Fanuc TP program (LS listing): S003.LS

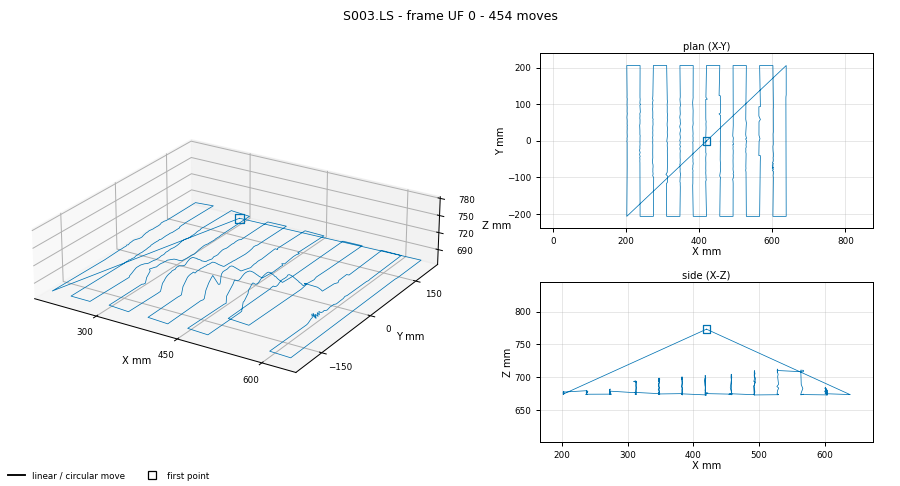
[picture p0: tool path of S003.LS in frame UF 0, 454 of 454 moves have a stored position in this frame; points joined in program order, loops and branches not executed]
/PROG  S003.LS
/ATTR
OWNER       = MNEDITOR;
COMMENT     = "";
PROG_SIZE   = 636;
CREATE      = DATE 23-01-07  TIME 11:59:14;
MODIFIED    = DATE 23-01-07  TIME 12:02:18;
FILE_NAME   = ;
VERSION     = 0;
LINE_COUNT  = 4;
MEMORY_SIZE = 992;
PROTECT     = READ_WRITE;
TCD:  STACK_SIZE    = 0,
      TASK_PRIORITY = 50,
      TIME_SLICE    = 0,
      BUSY_LAMP_OFF = 0,
      ABORT_REQUEST = 0,
      PAUSE_REQUEST = 0;
DEFAULT_GROUP    = 1,*,*,*,*;
CONTROL_CODE     = 00000000 00000000;
/MN
   1:J P[1] 100% FINE    ;
   2:L P[2] 300mm/sec CNT100    ;
   3:L P[3] 300mm/sec CNT100    ;
   4:L P[4] 300mm/sec CNT100    ;
   5:L P[5] 300mm/sec CNT100    ;
   6:L P[6] 300mm/sec CNT100    ;
   7:L P[7] 300mm/sec CNT100    ;
   8:L P[8] 300mm/sec CNT100    ;
   9:L P[9] 300mm/sec CNT100    ;
   10:L P[10] 300mm/sec CNT100    ;
   11:L P[11] 300mm/sec CNT100    ;
   12:L P[12] 300mm/sec CNT100    ;
   13:L P[13] 300mm/sec CNT100    ;
   14:L P[14] 300mm/sec CNT100    ;
   15:L P[15] 300mm/sec CNT100    ;
   16:L P[16] 300mm/sec CNT100    ;
   17:L P[17] 300mm/sec CNT100    ;
   18:L P[18] 300mm/sec CNT100    ;
   19:L P[19] 300mm/sec CNT100    ;
   20:L P[20] 300mm/sec CNT100    ;
   21:L P[21] 300mm/sec CNT100    ;
   22:L P[22] 300mm/sec CNT100    ;
   23:L P[23] 300mm/sec CNT100    ;
   24:L P[24] 300mm/sec CNT100    ;
   25:L P[25] 300mm/sec CNT100    ;
   26:L P[26] 300mm/sec CNT100    ;
   27:L P[27] 300mm/sec CNT100    ;
   28:L P[28] 300mm/sec CNT100    ;
   29:L P[29] 300mm/sec CNT100    ;
   30:L P[30] 300mm/sec CNT100    ;
   31:L P[31] 300mm/sec CNT100    ;
   32:L P[32] 300mm/sec CNT100    ;
   33:L P[33] 300mm/sec CNT100    ;
   34:L P[34] 300mm/sec CNT100    ;
   35:L P[35] 300mm/sec CNT100    ;
   36:L P[36] 300mm/sec CNT100    ;
   37:L P[37] 300mm/sec CNT100    ;
   38:L P[38] 300mm/sec CNT100    ;
   39:L P[39] 300mm/sec CNT100    ;
   40:L P[40] 300mm/sec CNT100    ;
   41:L P[41] 300mm/sec CNT100    ;
   42:L P[42] 300mm/sec CNT100    ;
   43:L P[43] 300mm/sec CNT100    ;
   44:L P[44] 300mm/sec CNT100    ;
   45:L P[45] 300mm/sec CNT100    ;
   46:L P[46] 300mm/sec CNT100    ;
   47:L P[47] 300mm/sec CNT100    ;
   48:L P[48] 300mm/sec CNT100    ;
   49:L P[49] 300mm/sec CNT100    ;
   50:L P[50] 300mm/sec CNT100    ;
   51:L P[51] 300mm/sec CNT100    ;
   52:L P[52] 300mm/sec CNT100    ;
   53:L P[53] 300mm/sec CNT100    ;
   54:L P[54] 300mm/sec CNT100    ;
   55:L P[55] 300mm/sec CNT100    ;
   56:L P[56] 300mm/sec CNT100    ;
   57:L P[57] 300mm/sec CNT100    ;
   58:L P[58] 300mm/sec CNT100    ;
   59:L P[59] 300mm/sec CNT100    ;
   60:L P[60] 300mm/sec CNT100    ;
   61:L P[61] 300mm/sec CNT100    ;
   62:L P[62] 300mm/sec CNT100    ;
   63:L P[63] 300mm/sec CNT100    ;
   64:L P[64] 300mm/sec CNT100    ;
   65:L P[65] 300mm/sec CNT100    ;
   66:L P[66] 300mm/sec CNT100    ;
   67:L P[67] 300mm/sec CNT100    ;
   68:L P[68] 300mm/sec CNT100    ;
   69:L P[69] 300mm/sec CNT100    ;
   70:L P[70] 300mm/sec CNT100    ;
   71:L P[71] 300mm/sec CNT100    ;
   72:L P[72] 300mm/sec CNT100    ;
   73:L P[73] 300mm/sec CNT100    ;
   74:L P[74] 300mm/sec CNT100    ;
   75:L P[75] 300mm/sec CNT100    ;
   76:L P[76] 300mm/sec CNT100    ;
   77:L P[77] 300mm/sec CNT100    ;
   78:L P[78] 300mm/sec CNT100    ;
   79:L P[79] 300mm/sec CNT100    ;
   80:L P[80] 300mm/sec CNT100    ;
   81:L P[81] 300mm/sec CNT100    ;
   82:L P[82] 300mm/sec CNT100    ;
   83:L P[83] 300mm/sec CNT100    ;
   84:L P[84] 300mm/sec CNT100    ;
   85:L P[85] 300mm/sec CNT100    ;
   86:L P[86] 300mm/sec CNT100    ;
   87:L P[87] 300mm/sec CNT100    ;
   88:L P[88] 300mm/sec CNT100    ;
   89:L P[89] 300mm/sec CNT100    ;
   90:L P[90] 300mm/sec CNT100    ;
   91:L P[91] 300mm/sec CNT100    ;
   92:L P[92] 300mm/sec CNT100    ;
   93:L P[93] 300mm/sec CNT100    ;
   94:L P[94] 300mm/sec CNT100    ;
   95:L P[95] 300mm/sec CNT100    ;
   96:L P[96] 300mm/sec CNT100    ;
   97:L P[97] 300mm/sec CNT100    ;
   98:L P[98] 300mm/sec CNT100    ;
   99:L P[99] 300mm/sec CNT100    ;
   100:L P[100] 300mm/sec CNT100    ;
   101:L P[101] 300mm/sec CNT100    ;
   102:L P[102] 300mm/sec CNT100    ;
   103:L P[103] 300mm/sec CNT100    ;
   104:L P[104] 300mm/sec CNT100    ;
   105:L P[105] 300mm/sec CNT100    ;
   106:L P[106] 300mm/sec CNT100    ;
   107:L P[107] 300mm/sec CNT100    ;
   108:L P[108] 300mm/sec CNT100    ;
   109:L P[109] 300mm/sec CNT100    ;
   110:L P[110] 300mm/sec CNT100    ;
   111:L P[111] 300mm/sec CNT100    ;
   112:L P[112] 300mm/sec CNT100    ;
   113:L P[113] 300mm/sec CNT100    ;
   114:L P[114] 300mm/sec CNT100    ;
   115:L P[115] 300mm/sec CNT100    ;
   116:L P[116] 300mm/sec CNT100    ;
   117:L P[117] 300mm/sec CNT100    ;
   118:L P[118] 300mm/sec CNT100    ;
   119:L P[119] 300mm/sec CNT100    ;
   120:L P[120] 300mm/sec CNT100    ;
   121:L P[121] 300mm/sec CNT100    ;
   122:L P[122] 300mm/sec CNT100    ;
   123:L P[123] 300mm/sec CNT100    ;
   124:L P[124] 300mm/sec CNT100    ;
   125:L P[125] 300mm/sec CNT100    ;
   126:L P[126] 300mm/sec CNT100    ;
   127:L P[127] 300mm/sec CNT100    ;
   128:L P[128] 300mm/sec CNT100    ;
   129:L P[129] 300mm/sec CNT100    ;
   130:L P[130] 300mm/sec CNT100    ;
   131:L P[131] 300mm/sec CNT100    ;
   132:L P[132] 300mm/sec CNT100    ;
   133:L P[133] 300mm/sec CNT100    ;
   134:L P[134] 300mm/sec CNT100    ;
   135:L P[135] 300mm/sec CNT100    ;
   136:L P[136] 300mm/sec CNT100    ;
   137:L P[137] 300mm/sec CNT100    ;
   138:L P[138] 300mm/sec CNT100    ;
   139:L P[139] 300mm/sec CNT100    ;
   140:L P[140] 300mm/sec CNT100    ;
   141:L P[141] 300mm/sec CNT100    ;
   142:L P[142] 300mm/sec CNT100    ;
   143:L P[143] 300mm/sec CNT100    ;
   144:L P[144] 300mm/sec CNT100    ;
   145:L P[145] 300mm/sec CNT100    ;
   146:L P[146] 300mm/sec CNT100    ;
   147:L P[147] 300mm/sec CNT100    ;
   148:L P[148] 300mm/sec CNT100    ;
   149:L P[149] 300mm/sec CNT100    ;
   150:L P[150] 300mm/sec CNT100    ;
   151:L P[151] 300mm/sec CNT100    ;
   152:L P[152] 300mm/sec CNT100    ;
   153:L P[153] 300mm/sec CNT100    ;
   154:L P[154] 300mm/sec CNT100    ;
   155:L P[155] 300mm/sec CNT100    ;
   156:L P[156] 300mm/sec CNT100    ;
   157:L P[157] 300mm/sec CNT100    ;
   158:L P[158] 300mm/sec CNT100    ;
   159:L P[159] 300mm/sec CNT100    ;
   160:L P[160] 300mm/sec CNT100    ;
   161:L P[161] 300mm/sec CNT100    ;
   162:L P[162] 300mm/sec CNT100    ;
   163:L P[163] 300mm/sec CNT100    ;
   164:L P[164] 300mm/sec CNT100    ;
   165:L P[165] 300mm/sec CNT100    ;
   166:L P[166] 300mm/sec CNT100    ;
   167:L P[167] 300mm/sec CNT100    ;
   168:L P[168] 300mm/sec CNT100    ;
   169:L P[169] 300mm/sec CNT100    ;
   170:L P[170] 300mm/sec CNT100    ;
   171:L P[171] 300mm/sec CNT100    ;
   172:L P[172] 300mm/sec CNT100    ;
   173:L P[173] 300mm/sec CNT100    ;
   174:L P[174] 300mm/sec CNT100    ;
   175:L P[175] 300mm/sec CNT100    ;
   176:L P[176] 300mm/sec CNT100    ;
   177:L P[177] 300mm/sec CNT100    ;
   178:L P[178] 300mm/sec CNT100    ;
   179:L P[179] 300mm/sec CNT100    ;
   180:L P[180] 300mm/sec CNT100    ;
   181:L P[181] 300mm/sec CNT100    ;
   182:L P[182] 300mm/sec CNT100    ;
   183:L P[183] 300mm/sec CNT100    ;
   184:L P[184] 300mm/sec CNT100    ;
   185:L P[185] 300mm/sec CNT100    ;
   186:L P[186] 300mm/sec CNT100    ;
   187:L P[187] 300mm/sec CNT100    ;
   188:L P[188] 300mm/sec CNT100    ;
   189:L P[189] 300mm/sec CNT100    ;
   190:L P[190] 300mm/sec CNT100    ;
   191:L P[191] 300mm/sec CNT100    ;
   192:L P[192] 300mm/sec CNT100    ;
   193:L P[193] 300mm/sec CNT100    ;
   194:L P[194] 300mm/sec CNT100    ;
   195:L P[195] 300mm/sec CNT100    ;
   196:L P[196] 300mm/sec CNT100    ;
   197:L P[197] 300mm/sec CNT100    ;
   198:L P[198] 300mm/sec CNT100    ;
   199:L P[199] 300mm/sec CNT100    ;
   200:L P[200] 300mm/sec CNT100    ;
   201:L P[201] 300mm/sec CNT100    ;
   202:L P[202] 300mm/sec CNT100    ;
   203:L P[203] 300mm/sec CNT100    ;
   204:L P[204] 300mm/sec CNT100    ;
   205:L P[205] 300mm/sec CNT100    ;
   206:L P[206] 300mm/sec CNT100    ;
   207:L P[207] 300mm/sec CNT100    ;
   208:L P[208] 300mm/sec CNT100    ;
   209:L P[209] 300mm/sec CNT100    ;
   210:L P[210] 300mm/sec CNT100    ;
   211:L P[211] 300mm/sec CNT100    ;
   212:L P[212] 300mm/sec CNT100    ;
   213:L P[213] 300mm/sec CNT100    ;
   214:L P[214] 300mm/sec CNT100    ;
   215:L P[215] 300mm/sec CNT100    ;
   216:L P[216] 300mm/sec CNT100    ;
   217:L P[217] 300mm/sec CNT100    ;
   218:L P[218] 300mm/sec CNT100    ;
   219:L P[219] 300mm/sec CNT100    ;
   220:L P[220] 300mm/sec CNT100    ;
   221:L P[221] 300mm/sec CNT100    ;
   222:L P[222] 300mm/sec CNT100    ;
   223:L P[223] 300mm/sec CNT100    ;
   224:L P[224] 300mm/sec CNT100    ;
   225:L P[225] 300mm/sec CNT100    ;
   226:L P[226] 300mm/sec CNT100    ;
   227:L P[227] 300mm/sec CNT100    ;
   228:L P[228] 300mm/sec CNT100    ;
   229:L P[229] 300mm/sec CNT100    ;
   230:L P[230] 300mm/sec CNT100    ;
   231:L P[231] 300mm/sec CNT100    ;
   232:L P[232] 300mm/sec CNT100    ;
   233:L P[233] 300mm/sec CNT100    ;
   234:L P[234] 300mm/sec CNT100    ;
   235:L P[235] 300mm/sec CNT100    ;
   236:L P[236] 300mm/sec CNT100    ;
   237:L P[237] 300mm/sec CNT100    ;
   238:L P[238] 300mm/sec CNT100    ;
   239:L P[239] 300mm/sec CNT100    ;
   240:L P[240] 300mm/sec CNT100    ;
   241:L P[241] 300mm/sec CNT100    ;
   242:L P[242] 300mm/sec CNT100    ;
   243:L P[243] 300mm/sec CNT100    ;
   244:L P[244] 300mm/sec CNT100    ;
   245:L P[245] 300mm/sec CNT100    ;
   246:L P[246] 300mm/sec CNT100    ;
   247:L P[247] 300mm/sec CNT100    ;
   248:L P[248] 300mm/sec CNT100    ;
   249:L P[249] 300mm/sec CNT100    ;
   250:L P[250] 300mm/sec CNT100    ;
   251:L P[251] 300mm/sec CNT100    ;
   252:L P[252] 300mm/sec CNT100    ;
   253:L P[253] 300mm/sec CNT100    ;
   254:L P[254] 300mm/sec CNT100    ;
   255:L P[255] 300mm/sec CNT100    ;
   256:L P[256] 300mm/sec CNT100    ;
   257:L P[257] 300mm/sec CNT100    ;
   258:L P[258] 300mm/sec CNT100    ;
   259:L P[259] 300mm/sec CNT100    ;
   260:L P[260] 300mm/sec CNT100    ;
   261:L P[261] 300mm/sec CNT100    ;
   262:L P[262] 300mm/sec CNT100    ;
   263:L P[263] 300mm/sec CNT100    ;
   264:L P[264] 300mm/sec CNT100    ;
   265:L P[265] 300mm/sec CNT100    ;
   266:L P[266] 300mm/sec CNT100    ;
   267:L P[267] 300mm/sec CNT100    ;
   268:L P[268] 300mm/sec CNT100    ;
   269:L P[269] 300mm/sec CNT100    ;
   270:L P[270] 300mm/sec CNT100    ;
   271:L P[271] 300mm/sec CNT100    ;
   272:L P[272] 300mm/sec CNT100    ;
   273:L P[273] 300mm/sec CNT100    ;
   274:L P[274] 300mm/sec CNT100    ;
   275:L P[275] 300mm/sec CNT100    ;
   276:L P[276] 300mm/sec CNT100    ;
   277:L P[277] 300mm/sec CNT100    ;
   278:L P[278] 300mm/sec CNT100    ;
   279:L P[279] 300mm/sec CNT100    ;
   280:L P[280] 300mm/sec CNT100    ;
   281:L P[281] 300mm/sec CNT100    ;
   282:L P[282] 300mm/sec CNT100    ;
   283:L P[283] 300mm/sec CNT100    ;
   284:L P[284] 300mm/sec CNT100    ;
   285:L P[285] 300mm/sec CNT100    ;
   286:L P[286] 300mm/sec CNT100    ;
   287:L P[287] 300mm/sec CNT100    ;
   288:L P[288] 300mm/sec CNT100    ;
   289:L P[289] 300mm/sec CNT100    ;
   290:L P[290] 300mm/sec CNT100    ;
   291:L P[291] 300mm/sec CNT100    ;
   292:L P[292] 300mm/sec CNT100    ;
   293:L P[293] 300mm/sec CNT100    ;
   294:L P[294] 300mm/sec CNT100    ;
   295:L P[295] 300mm/sec CNT100    ;
   296:L P[296] 300mm/sec CNT100    ;
   297:L P[297] 300mm/sec CNT100    ;
   298:L P[298] 300mm/sec CNT100    ;
   299:L P[299] 300mm/sec CNT100    ;
   300:L P[300] 300mm/sec CNT100    ;
   301:L P[301] 300mm/sec CNT100    ;
   302:L P[302] 300mm/sec CNT100    ;
   303:L P[303] 300mm/sec CNT100    ;
   304:L P[304] 300mm/sec CNT100    ;
   305:L P[305] 300mm/sec CNT100    ;
   306:L P[306] 300mm/sec CNT100    ;
   307:L P[307] 300mm/sec CNT100    ;
   308:L P[308] 300mm/sec CNT100    ;
   309:L P[309] 300mm/sec CNT100    ;
   310:L P[310] 300mm/sec CNT100    ;
   311:L P[311] 300mm/sec CNT100    ;
   312:L P[312] 300mm/sec CNT100    ;
   313:L P[313] 300mm/sec CNT100    ;
   314:L P[314] 300mm/sec CNT100    ;
   315:L P[315] 300mm/sec CNT100    ;
   316:L P[316] 300mm/sec CNT100    ;
   317:L P[317] 300mm/sec CNT100    ;
   318:L P[318] 300mm/sec CNT100    ;
   319:L P[319] 300mm/sec CNT100    ;
   320:L P[320] 300mm/sec CNT100    ;
   321:L P[321] 300mm/sec CNT100    ;
   322:L P[322] 300mm/sec CNT100    ;
   323:L P[323] 300mm/sec CNT100    ;
   324:L P[324] 300mm/sec CNT100    ;
   325:L P[325] 300mm/sec CNT100    ;
   326:L P[326] 300mm/sec CNT100    ;
   327:L P[327] 300mm/sec CNT100    ;
   328:L P[328] 300mm/sec CNT100    ;
   329:L P[329] 300mm/sec CNT100    ;
   330:L P[330] 300mm/sec CNT100    ;
   331:L P[331] 300mm/sec CNT100    ;
   332:L P[332] 300mm/sec CNT100    ;
   333:L P[333] 300mm/sec CNT100    ;
   334:L P[334] 300mm/sec CNT100    ;
   335:L P[335] 300mm/sec CNT100    ;
   336:L P[336] 300mm/sec CNT100    ;
   337:L P[337] 300mm/sec CNT100    ;
   338:L P[338] 300mm/sec CNT100    ;
   339:L P[339] 300mm/sec CNT100    ;
   340:L P[340] 300mm/sec CNT100    ;
   341:L P[341] 300mm/sec CNT100    ;
   342:L P[342] 300mm/sec CNT100    ;
   343:L P[343] 300mm/sec CNT100    ;
   344:L P[344] 300mm/sec CNT100    ;
   345:L P[345] 300mm/sec CNT100    ;
   346:L P[346] 300mm/sec CNT100    ;
   347:L P[347] 300mm/sec CNT100    ;
   348:L P[348] 300mm/sec CNT100    ;
   349:L P[349] 300mm/sec CNT100    ;
   350:L P[350] 300mm/sec CNT100    ;
   351:L P[351] 300mm/sec CNT100    ;
   352:L P[352] 300mm/sec CNT100    ;
   353:L P[353] 300mm/sec CNT100    ;
   354:L P[354] 300mm/sec CNT100    ;
   355:L P[355] 300mm/sec CNT100    ;
   356:L P[356] 300mm/sec CNT100    ;
   357:L P[357] 300mm/sec CNT100    ;
   358:L P[358] 300mm/sec CNT100    ;
   359:L P[359] 300mm/sec CNT100    ;
   360:L P[360] 300mm/sec CNT100    ;
   361:L P[361] 300mm/sec CNT100    ;
   362:L P[362] 300mm/sec CNT100    ;
   363:L P[363] 300mm/sec CNT100    ;
   364:L P[364] 300mm/sec CNT100    ;
   365:L P[365] 300mm/sec CNT100    ;
   366:L P[366] 300mm/sec CNT100    ;
   367:L P[367] 300mm/sec CNT100    ;
   368:L P[368] 300mm/sec CNT100    ;
   369:L P[369] 300mm/sec CNT100    ;
   370:L P[370] 300mm/sec CNT100    ;
   371:L P[371] 300mm/sec CNT100    ;
   372:L P[372] 300mm/sec CNT100    ;
   373:L P[373] 300mm/sec CNT100    ;
   374:L P[374] 300mm/sec CNT100    ;
   375:L P[375] 300mm/sec CNT100    ;
   376:L P[376] 300mm/sec CNT100    ;
   377:L P[377] 300mm/sec CNT100    ;
   378:L P[378] 300mm/sec CNT100    ;
   379:L P[379] 300mm/sec CNT100    ;
   380:L P[380] 300mm/sec CNT100    ;
   381:L P[381] 300mm/sec CNT100    ;
   382:L P[382] 300mm/sec CNT100    ;
   383:L P[383] 300mm/sec CNT100    ;
   384:L P[384] 300mm/sec CNT100    ;
   385:L P[385] 300mm/sec CNT100    ;
   386:L P[386] 300mm/sec CNT100    ;
   387:L P[387] 300mm/sec CNT100    ;
   388:L P[388] 300mm/sec CNT100    ;
   389:L P[389] 300mm/sec CNT100    ;
   390:L P[390] 300mm/sec CNT100    ;
   391:L P[391] 300mm/sec CNT100    ;
   392:L P[392] 300mm/sec CNT100    ;
   393:L P[393] 300mm/sec CNT100    ;
   394:L P[394] 300mm/sec CNT100    ;
   395:L P[395] 300mm/sec CNT100    ;
   396:L P[396] 300mm/sec CNT100    ;
   397:L P[397] 300mm/sec CNT100    ;
   398:L P[398] 300mm/sec CNT100    ;
   399:L P[399] 300mm/sec CNT100    ;
   400:L P[400] 300mm/sec CNT100    ;
   401:L P[401] 300mm/sec CNT100    ;
   402:L P[402] 300mm/sec CNT100    ;
   403:L P[403] 300mm/sec CNT100    ;
   404:L P[404] 300mm/sec CNT100    ;
   405:L P[405] 300mm/sec CNT100    ;
   406:L P[406] 300mm/sec CNT100    ;
   407:L P[407] 300mm/sec CNT100    ;
   408:L P[408] 300mm/sec CNT100    ;
   409:L P[409] 300mm/sec CNT100    ;
   410:L P[410] 300mm/sec CNT100    ;
   411:L P[411] 300mm/sec CNT100    ;
   412:L P[412] 300mm/sec CNT100    ;
   413:L P[413] 300mm/sec CNT100    ;
   414:L P[414] 300mm/sec CNT100    ;
   415:L P[415] 300mm/sec CNT100    ;
   416:L P[416] 300mm/sec CNT100    ;
   417:L P[417] 300mm/sec CNT100    ;
   418:L P[418] 300mm/sec CNT100    ;
   419:L P[419] 300mm/sec CNT100    ;
   420:L P[420] 300mm/sec CNT100    ;
   421:L P[421] 300mm/sec CNT100    ;
   422:L P[422] 300mm/sec CNT100    ;
   423:L P[423] 300mm/sec CNT100    ;
   424:L P[424] 300mm/sec CNT100    ;
   425:L P[425] 300mm/sec CNT100    ;
   426:L P[426] 300mm/sec CNT100    ;
   427:L P[427] 300mm/sec CNT100    ;
   428:L P[428] 300mm/sec CNT100    ;
   429:L P[429] 300mm/sec CNT100    ;
   430:L P[430] 300mm/sec CNT100    ;
   431:L P[431] 300mm/sec CNT100    ;
   432:L P[432] 300mm/sec CNT100    ;
   433:L P[433] 300mm/sec CNT100    ;
   434:L P[434] 300mm/sec CNT100    ;
   435:L P[435] 300mm/sec CNT100    ;
   436:L P[436] 300mm/sec CNT100    ;
   437:L P[437] 300mm/sec CNT100    ;
   438:L P[438] 300mm/sec CNT100    ;
   439:L P[439] 300mm/sec CNT100    ;
   440:L P[440] 300mm/sec CNT100    ;
   441:L P[441] 300mm/sec CNT100    ;
   442:L P[442] 300mm/sec CNT100    ;
   443:L P[443] 300mm/sec CNT100    ;
   444:L P[444] 300mm/sec CNT100    ;
   445:L P[445] 300mm/sec CNT100    ;
   446:L P[446] 300mm/sec CNT100    ;
   447:L P[447] 300mm/sec CNT100    ;
   448:L P[448] 300mm/sec CNT100    ;
   449:L P[449] 300mm/sec CNT100    ;
   450:L P[450] 300mm/sec CNT100    ;
   451:L P[451] 300mm/sec CNT100    ;
   452:L P[452] 300mm/sec CNT100    ;
   453:L P[453] 300mm/sec CNT100    ;
   454:L P[454] 300mm/sec CNT100    ;
/POS
P[1]{
   GP1:
    UF : 0, UT : 6,      CONFIG : 'N U T, 0, 0, 0',
    X =  420.000  mm,    Y =   0.000  mm,    Z =   773.173  mm,
    W =  -180.000 deg,    P =   0.000 deg,    R =   0.000 deg
};
P[2]{
   GP1:
    UF : 0, UT : 6,      CONFIG : 'N U T, 0, 0, 0',
    X =  638.117  mm,    Y =   206.397  mm,    Z =   673.755  mm,
    W =  -180.000 deg,    P =   0.000 deg,    R =   0.000 deg
};
P[3]{
   GP1:
    UF : 0, UT : 6,      CONFIG : 'N U T, 0, 0, 0',
    X =  638.117  mm,    Y =   125.921  mm,    Z =   673.755  mm,
    W =  -180.402 deg,    P =   0.007 deg,    R =   -1.000 deg
};
P[4]{
   GP1:
    UF : 0, UT : 6,      CONFIG : 'N U T, 0, 0, 0',
    X =  637.395  mm,    Y =   120.900  mm,    Z =   673.755  mm,
    W =  -180.370 deg,    P =   0.006 deg,    R =   -1.000 deg
};
P[5]{
   GP1:
    UF : 0, UT : 6,      CONFIG : 'N U T, 0, 0, 0',
    X =  637.281  mm,    Y =   114.689  mm,    Z =   673.804  mm,
    W =  -180.188 deg,    P =   0.003 deg,    R =   -1.000 deg
};
P[6]{
   GP1:
    UF : 0, UT : 6,      CONFIG : 'N U T, 0, 0, 0',
    X =  638.117  mm,    Y =   -206.397  mm,    Z =   673.804  mm,
    W =  -180.000 deg,    P =   0.000 deg,    R =   0.000 deg
};
P[7]{
   GP1:
    UF : 0, UT : 6,      CONFIG : 'N U T, 0, 0, 0',
    X =  601.764  mm,    Y =   -206.397  mm,    Z =   675.061  mm,
    W =  -180.000 deg,    P =   0.000 deg,    R =   0.000 deg
};
P[8]{
   GP1:
    UF : 0, UT : 6,      CONFIG : 'N U T, 0, 0, 0',
    X =  603.063  mm,    Y =   -100.441  mm,    Z =   675.061  mm,
    W =  -181.575 deg,    P =   0.025 deg,    R =   -0.915 deg
};
P[9]{
   GP1:
    UF : 0, UT : 6,      CONFIG : 'N U T, 0, 0, 0',
    X =  602.352  mm,    Y =   -94.987  mm,    Z =   675.061  mm,
    W =  -179.589 deg,    P =   -0.007 deg,    R =   -0.926 deg
};
P[10]{
   GP1:
    UF : 0, UT : 6,      CONFIG : 'N U T, 0, 0, 0',
    X =  603.394  mm,    Y =   -87.376  mm,    Z =   680.006  mm,
    W =  -176.777 deg,    P =   -0.052 deg,    R =   -0.928 deg
};
P[11]{
   GP1:
    UF : 0, UT : 6,      CONFIG : 'N U T, 0, 0, 0',
    X =  603.228  mm,    Y =   -83.336  mm,    Z =   680.501  mm,
    W =  -175.289 deg,    P =   -0.077 deg,    R =   -0.931 deg
};
P[12]{
   GP1:
    UF : 0, UT : 6,      CONFIG : 'N U T, 0, 0, 0',
    X =  600.513  mm,    Y =   -80.897  mm,    Z =   684.490  mm,
    W =  -173.913 deg,    P =   -0.100 deg,    R =   -0.933 deg
};
P[13]{
   GP1:
    UF : 0, UT : 6,      CONFIG : 'N U T, 0, 0, 0',
    X =  603.162  mm,    Y =   -78.266  mm,    Z =   679.693  mm,
    W =  -173.089 deg,    P =   -0.113 deg,    R =   -0.929 deg
};
P[14]{
   GP1:
    UF : 0, UT : 6,      CONFIG : 'N U T, 0, 0, 0',
    X =  599.922  mm,    Y =   -75.857  mm,    Z =   683.697  mm,
    W =  -172.461 deg,    P =   -0.124 deg,    R =   -0.935 deg
};
P[15]{
   GP1:
    UF : 0, UT : 6,      CONFIG : 'N U T, 0, 0, 0',
    X =  603.955  mm,    Y =   -74.066  mm,    Z =   677.460  mm,
    W =  -172.156 deg,    P =   -0.128 deg,    R =   -0.926 deg
};
P[16]{
   GP1:
    UF : 0, UT : 6,      CONFIG : 'N U T, 0, 0, 0',
    X =  599.977  mm,    Y =   -71.667  mm,    Z =   675.988  mm,
    W =  -171.721 deg,    P =   -0.136 deg,    R =   -0.932 deg
};
P[17]{
   GP1:
    UF : 0, UT : 6,      CONFIG : 'N U T, 0, 0, 0',
    X =  602.967  mm,    Y =   -71.637  mm,    Z =   673.990  mm,
    W =  -171.769 deg,    P =   -0.134 deg,    R =   -0.927 deg
};
P[18]{
   GP1:
    UF : 0, UT : 6,      CONFIG : 'N U T, 0, 0, 0',
    X =  599.805  mm,    Y =   -68.008  mm,    Z =   678.688  mm,
    W =  -171.113 deg,    P =   -0.146 deg,    R =   -0.934 deg
};
P[19]{
   GP1:
    UF : 0, UT : 6,      CONFIG : 'N U T, 0, 0, 0',
    X =  603.165  mm,    Y =   -65.813  mm,    Z =   675.136  mm,
    W =  -170.890 deg,    P =   -0.149 deg,    R =   -0.929 deg
};
P[20]{
   GP1:
    UF : 0, UT : 6,      CONFIG : 'N U T, 0, 0, 0',
    X =  600.149  mm,    Y =   -63.289  mm,    Z =   679.687  mm,
    W =  -170.781 deg,    P =   -0.151 deg,    R =   -0.933 deg
};
P[21]{
   GP1:
    UF : 0, UT : 6,      CONFIG : 'N U T, 0, 0, 0',
    X =  603.067  mm,    Y =   -61.873  mm,    Z =   676.004  mm,
    W =  -170.640 deg,    P =   -0.153 deg,    R =   -0.929 deg
};
P[22]{
   GP1:
    UF : 0, UT : 6,      CONFIG : 'N U T, 0, 0, 0',
    X =  600.578  mm,    Y =   -59.045  mm,    Z =   680.056  mm,
    W =  -170.134 deg,    P =   -0.162 deg,    R =   -0.933 deg
};
P[23]{
   GP1:
    UF : 0, UT : 6,      CONFIG : 'N U T, 0, 0, 0',
    X =  602.693  mm,    Y =   -56.010  mm,    Z =   677.423  mm,
    W =  -169.832 deg,    P =   -0.167 deg,    R =   -0.932 deg
};
P[24]{
   GP1:
    UF : 0, UT : 6,      CONFIG : 'N U T, 0, 0, 0',
    X =  602.928  mm,    Y =   -50.751  mm,    Z =   676.680  mm,
    W =  -169.253 deg,    P =   -0.176 deg,    R =   -0.930 deg
};
P[25]{
   GP1:
    UF : 0, UT : 6,      CONFIG : 'N U T, 0, 0, 0',
    X =  602.383  mm,    Y =   -45.786  mm,    Z =   676.913  mm,
    W =  -168.905 deg,    P =   -0.182 deg,    R =   -0.930 deg
};
P[26]{
   GP1:
    UF : 0, UT : 6,      CONFIG : 'N U T, 0, 0, 0',
    X =  603.218  mm,    Y =   -42.439  mm,    Z =   675.578  mm,
    W =  -168.497 deg,    P =   -0.189 deg,    R =   -0.928 deg
};
P[27]{
   GP1:
    UF : 0, UT : 6,      CONFIG : 'N U T, 0, 0, 0',
    X =  603.471  mm,    Y =   -38.296  mm,    Z =   674.950  mm,
    W =  -168.315 deg,    P =   -0.192 deg,    R =   -0.928 deg
};
P[28]{
   GP1:
    UF : 0, UT : 6,      CONFIG : 'N U T, 0, 0, 0',
    X =  602.333  mm,    Y =   -27.315  mm,    Z =   675.409  mm,
    W =  -167.217 deg,    P =   -0.211 deg,    R =   -0.929 deg
};
P[29]{
   GP1:
    UF : 0, UT : 6,      CONFIG : 'N U T, 0, 0, 0',
    X =  602.170  mm,    Y =   -21.437  mm,    Z =   674.853  mm,
    W =  -166.723 deg,    P =   -0.219 deg,    R =   -0.929 deg
};
P[30]{
   GP1:
    UF : 0, UT : 6,      CONFIG : 'N U T, 0, 0, 0',
    X =  601.816  mm,    Y =   -15.269  mm,    Z =   674.641  mm,
    W =  -167.168 deg,    P =   -0.213 deg,    R =   -0.934 deg
};
P[31]{
   GP1:
    UF : 0, UT : 6,      CONFIG : 'N U T, 0, 0, 0',
    X =  602.854  mm,    Y =   -9.054  mm,    Z =   673.226  mm,
    W =  -167.032 deg,    P =   -0.216 deg,    R =   -0.937 deg
};
P[32]{
   GP1:
    UF : 0, UT : 6,      CONFIG : 'N U T, 0, 0, 0',
    X =  602.678  mm,    Y =   13.242  mm,    Z =   673.567  mm,
    W =  -168.194 deg,    P =   -0.200 deg,    R =   -0.958 deg
};
P[33]{
   GP1:
    UF : 0, UT : 6,      CONFIG : 'N U T, 0, 0, 0',
    X =  602.367  mm,    Y =   19.206  mm,    Z =   674.874  mm,
    W =  -168.576 deg,    P =   -0.195 deg,    R =   -0.964 deg
};
P[34]{
   GP1:
    UF : 0, UT : 6,      CONFIG : 'N U T, 0, 0, 0',
    X =  603.016  mm,    Y =   24.561  mm,    Z =   674.224  mm,
    W =  -169.632 deg,    P =   -0.178 deg,    R =   -0.973 deg
};
P[35]{
   GP1:
    UF : 0, UT : 6,      CONFIG : 'N U T, 0, 0, 0',
    X =  602.739  mm,    Y =   88.211  mm,    Z =   673.411  mm,
    W =  -177.459 deg,    P =   -0.044 deg,    R =   -0.999 deg
};
P[36]{
   GP1:
    UF : 0, UT : 6,      CONFIG : 'N U T, 0, 0, 0',
    X =  603.843  mm,    Y =   92.967  mm,    Z =   673.323  mm,
    W =  -178.252 deg,    P =   -0.030 deg,    R =   -1.000 deg
};
P[37]{
   GP1:
    UF : 0, UT : 6,      CONFIG : 'N U T, 0, 0, 0',
    X =  603.113  mm,    Y =   97.845  mm,    Z =   673.323  mm,
    W =  -178.837 deg,    P =   -0.020 deg,    R =   -1.000 deg
};
P[38]{
   GP1:
    UF : 0, UT : 6,      CONFIG : 'N U T, 0, 0, 0',
    X =  601.764  mm,    Y =   206.397  mm,    Z =   673.323  mm,
    W =  -180.000 deg,    P =   0.000 deg,    R =   0.000 deg
};
P[39]{
   GP1:
    UF : 0, UT : 6,      CONFIG : 'N U T, 0, 0, 0',
    X =  565.411  mm,    Y =   206.397  mm,    Z =   673.839  mm,
    W =  -180.000 deg,    P =   0.000 deg,    R =   0.000 deg
};
P[40]{
   GP1:
    UF : 0, UT : 6,      CONFIG : 'N U T, 0, 0, 0',
    X =  567.551  mm,    Y =   99.193  mm,    Z =   673.839  mm,
    W =  -177.882 deg,    P =   -0.037 deg,    R =   -0.999 deg
};
P[41]{
   GP1:
    UF : 0, UT : 6,      CONFIG : 'N U T, 0, 0, 0',
    X =  567.511  mm,    Y =   93.989  mm,    Z =   673.839  mm,
    W =  -176.857 deg,    P =   -0.055 deg,    R =   -0.998 deg
};
P[42]{
   GP1:
    UF : 0, UT : 6,      CONFIG : 'N U T, 0, 0, 0',
    X =  563.342  mm,    Y =   93.543  mm,    Z =   673.839  mm,
    W =  -176.694 deg,    P =   -0.058 deg,    R =   -0.998 deg
};
P[43]{
   GP1:
    UF : 0, UT : 6,      CONFIG : 'N U T, 0, 0, 0',
    X =  563.365  mm,    Y =   68.219  mm,    Z =   673.352  mm,
    W =  -172.588 deg,    P =   -0.129 deg,    R =   -0.992 deg
};
P[44]{
   GP1:
    UF : 0, UT : 6,      CONFIG : 'N U T, 0, 0, 0',
    X =  567.469  mm,    Y =   58.664  mm,    Z =   674.311  mm,
    W =  -170.736 deg,    P =   -0.161 deg,    R =   -0.987 deg
};
P[45]{
   GP1:
    UF : 0, UT : 6,      CONFIG : 'N U T, 0, 0, 0',
    X =  563.702  mm,    Y =   52.668  mm,    Z =   673.766  mm,
    W =  -169.108 deg,    P =   -0.189 deg,    R =   -0.982 deg
};
P[46]{
   GP1:
    UF : 0, UT : 6,      CONFIG : 'N U T, 0, 0, 0',
    X =  563.587  mm,    Y =   15.691  mm,    Z =   675.624  mm,
    W =  -166.091 deg,    P =   -0.239 deg,    R =   -0.966 deg
};
P[47]{
   GP1:
    UF : 0, UT : 6,      CONFIG : 'N U T, 0, 0, 0',
    X =  566.365  mm,    Y =   5.996  mm,    Z =   682.927  mm,
    W =  -166.177 deg,    P =   -0.237 deg,    R =   -0.964 deg
};
P[48]{
   GP1:
    UF : 0, UT : 6,      CONFIG : 'N U T, 0, 0, 0',
    X =  563.968  mm,    Y =   -0.670  mm,    Z =   689.010  mm,
    W =  -165.295 deg,    P =   -0.252 deg,    R =   -0.959 deg
};
P[49]{
   GP1:
    UF : 0, UT : 6,      CONFIG : 'N U T, 0, 0, 0',
    X =  563.260  mm,    Y =   -39.929  mm,    Z =   710.930  mm,
    W =  -168.980 deg,    P =   -0.189 deg,    R =   -0.971 deg
};
P[50]{
   GP1:
    UF : 0, UT : 6,      CONFIG : 'N U T, 0, 0, 0',
    X =  567.292  mm,    Y =   -40.087  mm,    Z =   710.593  mm,
    W =  -168.374 deg,    P =   -0.199 deg,    R =   -0.967 deg
};
P[51]{
   GP1:
    UF : 0, UT : 6,      CONFIG : 'N U T, 0, 0, 0',
    X =  567.515  mm,    Y =   -45.248  mm,    Z =   710.138  mm,
    W =  -169.489 deg,    P =   -0.180 deg,    R =   -0.971 deg
};
P[52]{
   GP1:
    UF : 0, UT : 6,      CONFIG : 'N U T, 0, 0, 0',
    X =  567.185  mm,    Y =   -56.758  mm,    Z =   708.454  mm,
    W =  -171.954 deg,    P =   -0.138 deg,    R =   -0.978 deg
};
P[53]{
   GP1:
    UF : 0, UT : 6,      CONFIG : 'N U T, 0, 0, 0',
    X =  565.411  mm,    Y =   -206.397  mm,    Z =   708.454  mm,
    W =  -180.000 deg,    P =   0.000 deg,    R =   0.000 deg
};
P[54]{
   GP1:
    UF : 0, UT : 6,      CONFIG : 'N U T, 0, 0, 0',
    X =  529.059  mm,    Y =   -206.397  mm,    Z =   710.391  mm,
    W =  -180.000 deg,    P =   0.000 deg,    R =   0.000 deg
};
P[55]{
   GP1:
    UF : 0, UT : 6,      CONFIG : 'N U T, 0, 0, 0',
    X =  528.137  mm,    Y =   -84.880  mm,    Z =   710.391  mm,
    W =  -184.157 deg,    P =   0.072 deg,    R =   -0.997 deg
};
P[56]{
   GP1:
    UF : 0, UT : 6,      CONFIG : 'N U T, 0, 0, 0',
    X =  527.271  mm,    Y =   -80.513  mm,    Z =   710.391  mm,
    W =  -182.312 deg,    P =   0.040 deg,    R =   -0.999 deg
};
P[57]{
   GP1:
    UF : 0, UT : 6,      CONFIG : 'N U T, 0, 0, 0',
    X =  528.058  mm,    Y =   -74.566  mm,    Z =   711.420  mm,
    W =  -178.490 deg,    P =   -0.026 deg,    R =   -0.999 deg
};
P[58]{
   GP1:
    UF : 0, UT : 6,      CONFIG : 'N U T, 0, 0, 0',
    X =  527.685  mm,    Y =   -70.653  mm,    Z =   708.617  mm,
    W =  -177.353 deg,    P =   -0.046 deg,    R =   -0.998 deg
};
P[59]{
   GP1:
    UF : 0, UT : 6,      CONFIG : 'N U T, 0, 0, 0',
    X =  527.958  mm,    Y =   -64.972  mm,    Z =   707.371  mm,
    W =  -176.288 deg,    P =   -0.065 deg,    R =   -0.997 deg
};
P[60]{
   GP1:
    UF : 0, UT : 6,      CONFIG : 'N U T, 0, 0, 0',
    X =  527.898  mm,    Y =   -60.462  mm,    Z =   707.900  mm,
    W =  -175.618 deg,    P =   -0.076 deg,    R =   -0.996 deg
};
P[61]{
   GP1:
    UF : 0, UT : 6,      CONFIG : 'N U T, 0, 0, 0',
    X =  527.932  mm,    Y =   -56.468  mm,    Z =   709.741  mm,
    W =  -174.796 deg,    P =   -0.091 deg,    R =   -0.995 deg
};
P[62]{
   GP1:
    UF : 0, UT : 6,      CONFIG : 'N U T, 0, 0, 0',
    X =  527.752  mm,    Y =   -50.557  mm,    Z =   711.373  mm,
    W =  -174.056 deg,    P =   -0.103 deg,    R =   -0.994 deg
};
P[63]{
   GP1:
    UF : 0, UT : 6,      CONFIG : 'N U T, 0, 0, 0',
    X =  527.740  mm,    Y =   -45.202  mm,    Z =   711.327  mm,
    W =  -173.076 deg,    P =   -0.120 deg,    R =   -0.992 deg
};
P[64]{
   GP1:
    UF : 0, UT : 6,      CONFIG : 'N U T, 0, 0, 0',
    X =  528.060  mm,    Y =   -39.889  mm,    Z =   711.222  mm,
    W =  -171.600 deg,    P =   -0.146 deg,    R =   -0.989 deg
};
P[65]{
   GP1:
    UF : 0, UT : 6,      CONFIG : 'N U T, 0, 0, 0',
    X =  528.383  mm,    Y =   -34.649  mm,    Z =   711.653  mm,
    W =  -170.247 deg,    P =   -0.169 deg,    R =   -0.985 deg
};
P[66]{
   GP1:
    UF : 0, UT : 6,      CONFIG : 'N U T, 0, 0, 0',
    X =  527.454  mm,    Y =   -30.102  mm,    Z =   712.576  mm,
    W =  -168.415 deg,    P =   -0.201 deg,    R =   -0.979 deg
};
P[67]{
   GP1:
    UF : 0, UT : 6,      CONFIG : 'N U T, 0, 0, 0',
    X =  527.761  mm,    Y =   -26.194  mm,    Z =   711.743  mm,
    W =  -167.340 deg,    P =   -0.219 deg,    R =   -0.975 deg
};
P[68]{
   GP1:
    UF : 0, UT : 6,      CONFIG : 'N U T, 0, 0, 0',
    X =  527.560  mm,    Y =   -19.767  mm,    Z =   707.736  mm,
    W =  -166.146 deg,    P =   -0.239 deg,    R =   -0.970 deg
};
P[69]{
   GP1:
    UF : 0, UT : 6,      CONFIG : 'N U T, 0, 0, 0',
    X =  528.855  mm,    Y =   -16.648  mm,    Z =   704.864  mm,
    W =  -165.626 deg,    P =   -0.248 deg,    R =   -0.968 deg
};
P[70]{
   GP1:
    UF : 0, UT : 6,      CONFIG : 'N U T, 0, 0, 0',
    X =  528.137  mm,    Y =   -11.612  mm,    Z =   700.747  mm,
    W =  -164.864 deg,    P =   -0.261 deg,    R =   -0.965 deg
};
P[71]{
   GP1:
    UF : 0, UT : 6,      CONFIG : 'N U T, 0, 0, 0',
    X =  529.469  mm,    Y =   1.028  mm,    Z =   689.346  mm,
    W =  -164.487 deg,    P =   -0.267 deg,    R =   -0.963 deg
};
P[72]{
   GP1:
    UF : 0, UT : 6,      CONFIG : 'N U T, 0, 0, 0',
    X =  526.954  mm,    Y =   5.533  mm,    Z =   686.079  mm,
    W =  -164.571 deg,    P =   -0.266 deg,    R =   -0.964 deg
};
P[73]{
   GP1:
    UF : 0, UT : 6,      CONFIG : 'N U T, 0, 0, 0',
    X =  529.720  mm,    Y =   7.403  mm,    Z =   683.675  mm,
    W =  -164.852 deg,    P =   -0.261 deg,    R =   -0.965 deg
};
P[74]{
   GP1:
    UF : 0, UT : 6,      CONFIG : 'N U T, 0, 0, 0',
    X =  528.024  mm,    Y =   12.251  mm,    Z =   680.024  mm,
    W =  -164.968 deg,    P =   -0.259 deg,    R =   -0.966 deg
};
P[75]{
   GP1:
    UF : 0, UT : 6,      CONFIG : 'N U T, 0, 0, 0',
    X =  527.279  mm,    Y =   18.065  mm,    Z =   675.188  mm,
    W =  -164.925 deg,    P =   -0.260 deg,    R =   -0.966 deg
};
P[76]{
   GP1:
    UF : 0, UT : 6,      CONFIG : 'N U T, 0, 0, 0',
    X =  529.140  mm,    Y =   49.330  mm,    Z =   673.761  mm,
    W =  -167.588 deg,    P =   -0.215 deg,    R =   -0.977 deg
};
P[77]{
   GP1:
    UF : 0, UT : 6,      CONFIG : 'N U T, 0, 0, 0',
    X =  528.581  mm,    Y =   53.296  mm,    Z =   674.289  mm,
    W =  -168.387 deg,    P =   -0.201 deg,    R =   -0.979 deg
};
P[78]{
   GP1:
    UF : 0, UT : 6,      CONFIG : 'N U T, 0, 0, 0',
    X =  527.430  mm,    Y =   59.423  mm,    Z =   674.187  mm,
    W =  -169.809 deg,    P =   -0.177 deg,    R =   -0.984 deg
};
P[79]{
   GP1:
    UF : 0, UT : 6,      CONFIG : 'N U T, 0, 0, 0',
    X =  527.840  mm,    Y =   99.431  mm,    Z =   673.588  mm,
    W =  -177.925 deg,    P =   -0.036 deg,    R =   -0.999 deg
};
P[80]{
   GP1:
    UF : 0, UT : 6,      CONFIG : 'N U T, 0, 0, 0',
    X =  529.059  mm,    Y =   206.397  mm,    Z =   673.588  mm,
    W =  -180.000 deg,    P =   0.000 deg,    R =   0.000 deg
};
P[81]{
   GP1:
    UF : 0, UT : 6,      CONFIG : 'N U T, 0, 0, 0',
    X =  492.706  mm,    Y =   206.397  mm,    Z =   673.224  mm,
    W =  -180.000 deg,    P =   0.000 deg,    R =   0.000 deg
};
P[82]{
   GP1:
    UF : 0, UT : 6,      CONFIG : 'N U T, 0, 0, 0',
    X =  493.063  mm,    Y =   59.174  mm,    Z =   673.224  mm,
    W =  -170.941 deg,    P =   -0.157 deg,    R =   -0.987 deg
};
P[83]{
   GP1:
    UF : 0, UT : 6,      CONFIG : 'N U T, 0, 0, 0',
    X =  493.364  mm,    Y =   47.660  mm,    Z =   673.369  mm,
    W =  -168.705 deg,    P =   -0.196 deg,    R =   -0.980 deg
};
P[84]{
   GP1:
    UF : 0, UT : 6,      CONFIG : 'N U T, 0, 0, 0',
    X =  493.200  mm,    Y =   42.386  mm,    Z =   673.333  mm,
    W =  -168.047 deg,    P =   -0.207 deg,    R =   -0.978 deg
};
P[85]{
   GP1:
    UF : 0, UT : 6,      CONFIG : 'N U T, 0, 0, 0',
    X =  491.848  mm,    Y =   13.497  mm,    Z =   673.891  mm,
    W =  -166.428 deg,    P =   -0.234 deg,    R =   -0.971 deg
};
P[86]{
   GP1:
    UF : 0, UT : 6,      CONFIG : 'N U T, 0, 0, 0',
    X =  493.492  mm,    Y =   8.302  mm,    Z =   677.358  mm,
    W =  -166.262 deg,    P =   -0.237 deg,    R =   -0.971 deg
};
P[87]{
   GP1:
    UF : 0, UT : 6,      CONFIG : 'N U T, 0, 0, 0',
    X =  493.005  mm,    Y =   2.566  mm,    Z =   682.236  mm,
    W =  -166.504 deg,    P =   -0.233 deg,    R =   -0.971 deg
};
P[88]{
   GP1:
    UF : 0, UT : 6,      CONFIG : 'N U T, 0, 0, 0',
    X =  492.446  mm,    Y =   -3.751  mm,    Z =   687.937  mm,
    W =  -166.917 deg,    P =   -0.226 deg,    R =   -0.973 deg
};
P[89]{
   GP1:
    UF : 0, UT : 6,      CONFIG : 'N U T, 0, 0, 0',
    X =  494.284  mm,    Y =   -9.420  mm,    Z =   692.851  mm,
    W =  -167.281 deg,    P =   -0.220 deg,    R =   -0.974 deg
};
P[90]{
   GP1:
    UF : 0, UT : 6,      CONFIG : 'N U T, 0, 0, 0',
    X =  491.887  mm,    Y =   -10.032  mm,    Z =   693.659  mm,
    W =  -167.546 deg,    P =   -0.215 deg,    R =   -0.975 deg
};
P[91]{
   GP1:
    UF : 0, UT : 6,      CONFIG : 'N U T, 0, 0, 0',
    X =  492.978  mm,    Y =   -15.260  mm,    Z =   698.052  mm,
    W =  -168.371 deg,    P =   -0.201 deg,    R =   -0.977 deg
};
P[92]{
   GP1:
    UF : 0, UT : 6,      CONFIG : 'N U T, 0, 0, 0',
    X =  492.496  mm,    Y =   -20.661  mm,    Z =   702.730  mm,
    W =  -169.190 deg,    P =   -0.187 deg,    R =   -0.980 deg
};
P[93]{
   GP1:
    UF : 0, UT : 6,      CONFIG : 'N U T, 0, 0, 0',
    X =  493.128  mm,    Y =   -26.742  mm,    Z =   707.142  mm,
    W =  -169.845 deg,    P =   -0.176 deg,    R =   -0.981 deg
};
P[94]{
   GP1:
    UF : 0, UT : 6,      CONFIG : 'N U T, 0, 0, 0',
    X =  493.183  mm,    Y =   -31.278  mm,    Z =   709.544  mm,
    W =  -170.326 deg,    P =   -0.167 deg,    R =   -0.982 deg
};
P[95]{
   GP1:
    UF : 0, UT : 6,      CONFIG : 'N U T, 0, 0, 0',
    X =  493.021  mm,    Y =   -34.538  mm,    Z =   710.264  mm,
    W =  -170.859 deg,    P =   -0.158 deg,    R =   -0.983 deg
};
P[96]{
   GP1:
    UF : 0, UT : 6,      CONFIG : 'N U T, 0, 0, 0',
    X =  492.670  mm,    Y =   -40.584  mm,    Z =   709.566  mm,
    W =  -171.894 deg,    P =   -0.140 deg,    R =   -0.986 deg
};
P[97]{
   GP1:
    UF : 0, UT : 6,      CONFIG : 'N U T, 0, 0, 0',
    X =  492.889  mm,    Y =   -45.648  mm,    Z =   709.123  mm,
    W =  -172.641 deg,    P =   -0.128 deg,    R =   -0.987 deg
};
P[98]{
   GP1:
    UF : 0, UT : 6,      CONFIG : 'N U T, 0, 0, 0',
    X =  492.649  mm,    Y =   -49.802  mm,    Z =   707.748  mm,
    W =  -173.384 deg,    P =   -0.115 deg,    R =   -0.989 deg
};
P[99]{
   GP1:
    UF : 0, UT : 6,      CONFIG : 'N U T, 0, 0, 0',
    X =  492.607  mm,    Y =   -54.006  mm,    Z =   706.142  mm,
    W =  -173.992 deg,    P =   -0.104 deg,    R =   -0.990 deg
};
P[100]{
   GP1:
    UF : 0, UT : 6,      CONFIG : 'N U T, 0, 0, 0',
    X =  492.607  mm,    Y =   -58.538  mm,    Z =   703.732  mm,
    W =  -174.716 deg,    P =   -0.092 deg,    R =   -0.991 deg
};
P[101]{
   GP1:
    UF : 0, UT : 6,      CONFIG : 'N U T, 0, 0, 0',
    X =  492.792  mm,    Y =   -63.988  mm,    Z =   702.458  mm,
    W =  -175.148 deg,    P =   -0.084 deg,    R =   -0.991 deg
};
P[102]{
   GP1:
    UF : 0, UT : 6,      CONFIG : 'N U T, 0, 0, 0',
    X =  492.933  mm,    Y =   -69.858  mm,    Z =   703.754  mm,
    W =  -176.054 deg,    P =   -0.068 deg,    R =   -0.992 deg
};
P[103]{
   GP1:
    UF : 0, UT : 6,      CONFIG : 'N U T, 0, 0, 0',
    X =  492.564  mm,    Y =   -76.730  mm,    Z =   708.838  mm,
    W =  -178.034 deg,    P =   -0.034 deg,    R =   -0.993 deg
};
P[104]{
   GP1:
    UF : 0, UT : 6,      CONFIG : 'N U T, 0, 0, 0',
    X =  492.938  mm,    Y =   -80.984  mm,    Z =   708.481  mm,
    W =  -179.371 deg,    P =   -0.011 deg,    R =   -0.993 deg
};
P[105]{
   GP1:
    UF : 0, UT : 6,      CONFIG : 'N U T, 0, 0, 0',
    X =  493.711  mm,    Y =   -85.924  mm,    Z =   705.991  mm,
    W =  -180.870 deg,    P =   0.015 deg,    R =   -0.993 deg
};
P[106]{
   GP1:
    UF : 0, UT : 6,      CONFIG : 'N U T, 0, 0, 0',
    X =  492.807  mm,    Y =   -90.193  mm,    Z =   701.890  mm,
    W =  -182.498 deg,    P =   0.043 deg,    R =   -0.992 deg
};
P[107]{
   GP1:
    UF : 0, UT : 6,      CONFIG : 'N U T, 0, 0, 0',
    X =  494.490  mm,    Y =   -94.313  mm,    Z =   698.418  mm,
    W =  -183.847 deg,    P =   0.067 deg,    R =   -0.991 deg
};
P[108]{
   GP1:
    UF : 0, UT : 6,      CONFIG : 'N U T, 0, 0, 0',
    X =  492.861  mm,    Y =   -102.879  mm,    Z =   688.250  mm,
    W =  -187.159 deg,    P =   0.124 deg,    R =   -0.985 deg
};
P[109]{
   GP1:
    UF : 0, UT : 6,      CONFIG : 'N U T, 0, 0, 0',
    X =  491.609  mm,    Y =   -103.985  mm,    Z =   686.572  mm,
    W =  -187.801 deg,    P =   0.135 deg,    R =   -0.983 deg
};
P[110]{
   GP1:
    UF : 0, UT : 6,      CONFIG : 'N U T, 0, 0, 0',
    X =  492.581  mm,    Y =   -109.839  mm,    Z =   673.582  mm,
    W =  -191.567 deg,    P =   0.199 deg,    R =   -0.973 deg
};
P[111]{
   GP1:
    UF : 0, UT : 6,      CONFIG : 'N U T, 0, 0, 0',
    X =  492.950  mm,    Y =   -116.474  mm,    Z =   673.582  mm,
    W =  -194.761 deg,    P =   0.253 deg,    R =   -0.960 deg
};
P[112]{
   GP1:
    UF : 0, UT : 6,      CONFIG : 'N U T, 0, 0, 0',
    X =  492.706  mm,    Y =   -206.397  mm,    Z =   673.582  mm,
    W =  -180.000 deg,    P =   0.000 deg,    R =   0.000 deg
};
P[113]{
   GP1:
    UF : 0, UT : 6,      CONFIG : 'N U T, 0, 0, 0',
    X =  456.353  mm,    Y =   -206.397  mm,    Z =   675.052  mm,
    W =  -180.000 deg,    P =   0.000 deg,    R =   0.000 deg
};
P[114]{
   GP1:
    UF : 0, UT : 6,      CONFIG : 'N U T, 0, 0, 0',
    X =  457.648  mm,    Y =   -105.748  mm,    Z =   675.052  mm,
    W =  -188.590 deg,    P =   0.149 deg,    R =   -0.985 deg
};
P[115]{
   GP1:
    UF : 0, UT : 6,      CONFIG : 'N U T, 0, 0, 0',
    X =  458.532  mm,    Y =   -100.866  mm,    Z =   675.052  mm,
    W =  -186.195 deg,    P =   0.107 deg,    R =   -0.990 deg
};
P[116]{
   GP1:
    UF : 0, UT : 6,      CONFIG : 'N U T, 0, 0, 0',
    X =  456.150  mm,    Y =   -95.833  mm,    Z =   684.503  mm,
    W =  -184.503 deg,    P =   0.078 deg,    R =   -0.993 deg
};
P[117]{
   GP1:
    UF : 0, UT : 6,      CONFIG : 'N U T, 0, 0, 0',
    X =  458.396  mm,    Y =   -80.559  mm,    Z =   699.788  mm,
    W =  -179.881 deg,    P =   -0.002 deg,    R =   -0.995 deg
};
P[118]{
   GP1:
    UF : 0, UT : 6,      CONFIG : 'N U T, 0, 0, 0',
    X =  457.935  mm,    Y =   -75.225  mm,    Z =   704.692  mm,
    W =  -179.256 deg,    P =   -0.013 deg,    R =   -0.995 deg
};
P[119]{
   GP1:
    UF : 0, UT : 6,      CONFIG : 'N U T, 0, 0, 0',
    X =  457.894  mm,    Y =   -66.885  mm,    Z =   700.049  mm,
    W =  -177.104 deg,    P =   -0.050 deg,    R =   -0.994 deg
};
P[120]{
   GP1:
    UF : 0, UT : 6,      CONFIG : 'N U T, 0, 0, 0',
    X =  458.177  mm,    Y =   -61.872  mm,    Z =   699.506  mm,
    W =  -176.264 deg,    P =   -0.065 deg,    R =   -0.993 deg
};
P[121]{
   GP1:
    UF : 0, UT : 6,      CONFIG : 'N U T, 0, 0, 0',
    X =  457.757  mm,    Y =   -57.154  mm,    Z =   700.089  mm,
    W =  -175.401 deg,    P =   -0.080 deg,    R =   -0.993 deg
};
P[122]{
   GP1:
    UF : 0, UT : 6,      CONFIG : 'N U T, 0, 0, 0',
    X =  457.473  mm,    Y =   -52.008  mm,    Z =   701.919  mm,
    W =  -174.453 deg,    P =   -0.096 deg,    R =   -0.991 deg
};
P[123]{
   GP1:
    UF : 0, UT : 6,      CONFIG : 'N U T, 0, 0, 0',
    X =  457.490  mm,    Y =   -45.362  mm,    Z =   703.943  mm,
    W =  -173.561 deg,    P =   -0.112 deg,    R =   -0.990 deg
};
P[124]{
   GP1:
    UF : 0, UT : 6,      CONFIG : 'N U T, 0, 0, 0',
    X =  457.512  mm,    Y =   -41.023  mm,    Z =   704.173  mm,
    W =  -172.799 deg,    P =   -0.125 deg,    R =   -0.989 deg
};
P[125]{
   GP1:
    UF : 0, UT : 6,      CONFIG : 'N U T, 0, 0, 0',
    X =  457.545  mm,    Y =   -36.202  mm,    Z =   703.779  mm,
    W =  -172.287 deg,    P =   -0.134 deg,    R =   -0.988 deg
};
P[126]{
   GP1:
    UF : 0, UT : 6,      CONFIG : 'N U T, 0, 0, 0',
    X =  457.808  mm,    Y =   -30.365  mm,    Z =   702.586  mm,
    W =  -171.760 deg,    P =   -0.143 deg,    R =   -0.986 deg
};
P[127]{
   GP1:
    UF : 0, UT : 6,      CONFIG : 'N U T, 0, 0, 0',
    X =  457.273  mm,    Y =   -25.142  mm,    Z =   699.970  mm,
    W =  -171.267 deg,    P =   -0.151 deg,    R =   -0.986 deg
};
P[128]{
   GP1:
    UF : 0, UT : 6,      CONFIG : 'N U T, 0, 0, 0',
    X =  457.721  mm,    Y =   -19.721  mm,    Z =   696.435  mm,
    W =  -170.747 deg,    P =   -0.160 deg,    R =   -0.984 deg
};
P[129]{
   GP1:
    UF : 0, UT : 6,      CONFIG : 'N U T, 0, 0, 0',
    X =  457.783  mm,    Y =   -15.345  mm,    Z =   693.099  mm,
    W =  -170.240 deg,    P =   -0.169 deg,    R =   -0.983 deg
};
P[130]{
   GP1:
    UF : 0, UT : 6,      CONFIG : 'N U T, 0, 0, 0',
    X =  457.858  mm,    Y =   -10.339  mm,    Z =   688.965  mm,
    W =  -169.968 deg,    P =   -0.174 deg,    R =   -0.982 deg
};
P[131]{
   GP1:
    UF : 0, UT : 6,      CONFIG : 'N U T, 0, 0, 0',
    X =  457.925  mm,    Y =   -5.711  mm,    Z =   685.386  mm,
    W =  -169.216 deg,    P =   -0.187 deg,    R =   -0.980 deg
};
P[132]{
   GP1:
    UF : 0, UT : 6,      CONFIG : 'N U T, 0, 0, 0',
    X =  457.601  mm,    Y =   -0.702  mm,    Z =   681.348  mm,
    W =  -168.760 deg,    P =   -0.194 deg,    R =   -0.979 deg
};
P[133]{
   GP1:
    UF : 0, UT : 6,      CONFIG : 'N U T, 0, 0, 0',
    X =  458.050  mm,    Y =   3.209  mm,    Z =   678.802  mm,
    W =  -168.576 deg,    P =   -0.198 deg,    R =   -0.978 deg
};
P[134]{
   GP1:
    UF : 0, UT : 6,      CONFIG : 'N U T, 0, 0, 0',
    X =  458.110  mm,    Y =   7.497  mm,    Z =   675.797  mm,
    W =  -168.516 deg,    P =   -0.199 deg,    R =   -0.978 deg
};
P[135]{
   GP1:
    UF : 0, UT : 6,      CONFIG : 'N U T, 0, 0, 0',
    X =  458.340  mm,    Y =   42.386  mm,    Z =   673.333  mm,
    W =  -169.941 deg,    P =   -0.175 deg,    R =   -0.984 deg
};
P[136]{
   GP1:
    UF : 0, UT : 6,      CONFIG : 'N U T, 0, 0, 0',
    X =  458.375  mm,    Y =   48.931  mm,    Z =   673.761  mm,
    W =  -170.616 deg,    P =   -0.163 deg,    R =   -0.986 deg
};
P[137]{
   GP1:
    UF : 0, UT : 6,      CONFIG : 'N U T, 0, 0, 0',
    X =  458.403  mm,    Y =   53.740  mm,    Z =   673.769  mm,
    W =  -171.337 deg,    P =   -0.151 deg,    R =   -0.988 deg
};
P[138]{
   GP1:
    UF : 0, UT : 6,      CONFIG : 'N U T, 0, 0, 0',
    X =  458.457  mm,    Y =   64.061  mm,    Z =   674.349  mm,
    W =  -173.311 deg,    P =   -0.116 deg,    R =   -0.993 deg
};
P[139]{
   GP1:
    UF : 0, UT : 6,      CONFIG : 'N U T, 0, 0, 0',
    X =  458.456  mm,    Y =   69.915  mm,    Z =   673.735  mm,
    W =  -174.443 deg,    P =   -0.097 deg,    R =   -0.995 deg
};
P[140]{
   GP1:
    UF : 0, UT : 6,      CONFIG : 'N U T, 0, 0, 0',
    X =  454.274  mm,    Y =   74.039  mm,    Z =   674.244  mm,
    W =  -175.368 deg,    P =   -0.081 deg,    R =   -0.997 deg
};
P[141]{
   GP1:
    UF : 0, UT : 6,      CONFIG : 'N U T, 0, 0, 0',
    X =  458.320  mm,    Y =   76.221  mm,    Z =   673.972  mm,
    W =  -175.810 deg,    P =   -0.073 deg,    R =   -0.997 deg
};
P[142]{
   GP1:
    UF : 0, UT : 6,      CONFIG : 'N U T, 0, 0, 0',
    X =  458.401  mm,    Y =   93.737  mm,    Z =   675.688  mm,
    W =  -179.145 deg,    P =   -0.015 deg,    R =   -1.000 deg
};
P[143]{
   GP1:
    UF : 0, UT : 6,      CONFIG : 'N U T, 0, 0, 0',
    X =  458.067  mm,    Y =   104.309  mm,    Z =   676.194  mm,
    W =  -180.613 deg,    P =   0.011 deg,    R =   -1.000 deg
};
P[144]{
   GP1:
    UF : 0, UT : 6,      CONFIG : 'N U T, 0, 0, 0',
    X =  457.840  mm,    Y =   109.924  mm,    Z =   675.895  mm,
    W =  -180.821 deg,    P =   0.014 deg,    R =   -1.000 deg
};
P[145]{
   GP1:
    UF : 0, UT : 6,      CONFIG : 'N U T, 0, 0, 0',
    X =  457.868  mm,    Y =   114.816  mm,    Z =   675.665  mm,
    W =  -180.817 deg,    P =   0.014 deg,    R =   -1.000 deg
};
P[146]{
   GP1:
    UF : 0, UT : 6,      CONFIG : 'N U T, 0, 0, 0',
    X =  457.902  mm,    Y =   120.100  mm,    Z =   674.460  mm,
    W =  -180.794 deg,    P =   0.014 deg,    R =   -1.000 deg
};
P[147]{
   GP1:
    UF : 0, UT : 6,      CONFIG : 'N U T, 0, 0, 0',
    X =  457.918  mm,    Y =   123.526  mm,    Z =   674.460  mm,
    W =  -180.768 deg,    P =   0.013 deg,    R =   -1.000 deg
};
P[148]{
   GP1:
    UF : 0, UT : 6,      CONFIG : 'N U T, 0, 0, 0',
    X =  454.414  mm,    Y =   124.264  mm,    Z =   674.460  mm,
    W =  -180.807 deg,    P =   0.014 deg,    R =   -1.000 deg
};
P[149]{
   GP1:
    UF : 0, UT : 6,      CONFIG : 'N U T, 0, 0, 0',
    X =  456.353  mm,    Y =   206.397  mm,    Z =   674.460  mm,
    W =  -180.000 deg,    P =   0.000 deg,    R =   0.000 deg
};
P[150]{
   GP1:
    UF : 0, UT : 6,      CONFIG : 'N U T, 0, 0, 0',
    X =  420.000  mm,    Y =   206.397  mm,    Z =   675.256  mm,
    W =  -180.000 deg,    P =   0.000 deg,    R =   0.000 deg
};
P[151]{
   GP1:
    UF : 0, UT : 6,      CONFIG : 'N U T, 0, 0, 0',
    X =  418.399  mm,    Y =   125.053  mm,    Z =   675.256  mm,
    W =  -180.603 deg,    P =   0.011 deg,    R =   -1.000 deg
};
P[152]{
   GP1:
    UF : 0, UT : 6,      CONFIG : 'N U T, 0, 0, 0',
    X =  418.390  mm,    Y =   119.455  mm,    Z =   675.256  mm,
    W =  -180.625 deg,    P =   0.011 deg,    R =   -1.000 deg
};
P[153]{
   GP1:
    UF : 0, UT : 6,      CONFIG : 'N U T, 0, 0, 0',
    X =  422.168  mm,    Y =   114.208  mm,    Z =   676.285  mm,
    W =  -180.639 deg,    P =   0.011 deg,    R =   -1.000 deg
};
P[154]{
   GP1:
    UF : 0, UT : 6,      CONFIG : 'N U T, 0, 0, 0',
    X =  417.859  mm,    Y =   113.538  mm,    Z =   676.968  mm,
    W =  -180.622 deg,    P =   0.011 deg,    R =   -1.000 deg
};
P[155]{
   GP1:
    UF : 0, UT : 6,      CONFIG : 'N U T, 0, 0, 0',
    X =  417.969  mm,    Y =   108.835  mm,    Z =   677.015  mm,
    W =  -180.569 deg,    P =   0.010 deg,    R =   -1.000 deg
};
P[156]{
   GP1:
    UF : 0, UT : 6,      CONFIG : 'N U T, 0, 0, 0',
    X =  417.904  mm,    Y =   70.346  mm,    Z =   674.671  mm,
    W =  -175.299 deg,    P =   -0.082 deg,    R =   -0.997 deg
};
P[157]{
   GP1:
    UF : 0, UT : 6,      CONFIG : 'N U T, 0, 0, 0',
    X =  418.101  mm,    Y =   63.586  mm,    Z =   675.513  mm,
    W =  -174.239 deg,    P =   -0.100 deg,    R =   -0.995 deg
};
P[158]{
   GP1:
    UF : 0, UT : 6,      CONFIG : 'N U T, 0, 0, 0',
    X =  418.247  mm,    Y =   57.545  mm,    Z =   675.604  mm,
    W =  -173.455 deg,    P =   -0.114 deg,    R =   -0.993 deg
};
P[159]{
   GP1:
    UF : 0, UT : 6,      CONFIG : 'N U T, 0, 0, 0',
    X =  419.023  mm,    Y =   52.702  mm,    Z =   675.483  mm,
    W =  -172.734 deg,    P =   -0.126 deg,    R =   -0.992 deg
};
P[160]{
   GP1:
    UF : 0, UT : 6,      CONFIG : 'N U T, 0, 0, 0',
    X =  418.464  mm,    Y =   47.297  mm,    Z =   675.063  mm,
    W =  -172.071 deg,    P =   -0.138 deg,    R =   -0.990 deg
};
P[161]{
   GP1:
    UF : 0, UT : 6,      CONFIG : 'N U T, 0, 0, 0',
    X =  418.564  mm,    Y =   41.588  mm,    Z =   674.292  mm,
    W =  -171.770 deg,    P =   -0.143 deg,    R =   -0.990 deg
};
P[162]{
   GP1:
    UF : 0, UT : 6,      CONFIG : 'N U T, 0, 0, 0',
    X =  418.869  mm,    Y =   35.751  mm,    Z =   673.407  mm,
    W =  -171.449 deg,    P =   -0.149 deg,    R =   -0.989 deg
};
P[163]{
   GP1:
    UF : 0, UT : 6,      CONFIG : 'N U T, 0, 0, 0',
    X =  417.927  mm,    Y =   7.683  mm,    Z =   678.161  mm,
    W =  -169.422 deg,    P =   -0.183 deg,    R =   -0.983 deg
};
P[164]{
   GP1:
    UF : 0, UT : 6,      CONFIG : 'N U T, 0, 0, 0',
    X =  418.190  mm,    Y =   3.182  mm,    Z =   681.431  mm,
    W =  -169.497 deg,    P =   -0.182 deg,    R =   -0.983 deg
};
P[165]{
   GP1:
    UF : 0, UT : 6,      CONFIG : 'N U T, 0, 0, 0',
    X =  418.471  mm,    Y =   -1.500  mm,    Z =   684.982  mm,
    W =  -169.583 deg,    P =   -0.181 deg,    R =   -0.983 deg
};
P[166]{
   GP1:
    UF : 0, UT : 6,      CONFIG : 'N U T, 0, 0, 0',
    X =  417.934  mm,    Y =   -5.749  mm,    Z =   688.008  mm,
    W =  -169.855 deg,    P =   -0.176 deg,    R =   -0.984 deg
};
P[167]{
   GP1:
    UF : 0, UT : 6,      CONFIG : 'N U T, 0, 0, 0',
    X =  417.804  mm,    Y =   -16.378  mm,    Z =   695.758  mm,
    W =  -170.958 deg,    P =   -0.157 deg,    R =   -0.987 deg
};
P[168]{
   GP1:
    UF : 0, UT : 6,      CONFIG : 'N U T, 0, 0, 0',
    X =  418.035  mm,    Y =   -20.926  mm,    Z =   698.059  mm,
    W =  -171.374 deg,    P =   -0.150 deg,    R =   -0.988 deg
};
P[169]{
   GP1:
    UF : 0, UT : 6,      CONFIG : 'N U T, 0, 0, 0',
    X =  418.131  mm,    Y =   -25.615  mm,    Z =   699.096  mm,
    W =  -171.867 deg,    P =   -0.141 deg,    R =   -0.989 deg
};
P[170]{
   GP1:
    UF : 0, UT : 6,      CONFIG : 'N U T, 0, 0, 0',
    X =  418.060  mm,    Y =   -31.952  mm,    Z =   697.860  mm,
    W =  -172.567 deg,    P =   -0.129 deg,    R =   -0.991 deg
};
P[171]{
   GP1:
    UF : 0, UT : 6,      CONFIG : 'N U T, 0, 0, 0',
    X =  419.015  mm,    Y =   -34.875  mm,    Z =   698.344  mm,
    W =  -172.899 deg,    P =   -0.123 deg,    R =   -0.991 deg
};
P[172]{
   GP1:
    UF : 0, UT : 6,      CONFIG : 'N U T, 0, 0, 0',
    X =  417.917  mm,    Y =   -45.610  mm,    Z =   697.818  mm,
    W =  -174.424 deg,    P =   -0.097 deg,    R =   -0.994 deg
};
P[173]{
   GP1:
    UF : 0, UT : 6,      CONFIG : 'N U T, 0, 0, 0',
    X =  417.914  mm,    Y =   -50.211  mm,    Z =   695.324  mm,
    W =  -175.186 deg,    P =   -0.084 deg,    R =   -0.995 deg
};
P[174]{
   GP1:
    UF : 0, UT : 6,      CONFIG : 'N U T, 0, 0, 0',
    X =  417.921  mm,    Y =   -52.097  mm,    Z =   690.340  mm,
    W =  -175.487 deg,    P =   -0.079 deg,    R =   -0.996 deg
};
P[175]{
   GP1:
    UF : 0, UT : 6,      CONFIG : 'N U T, 0, 0, 0',
    X =  418.201  mm,    Y =   -53.556  mm,    Z =   684.107  mm,
    W =  -175.616 deg,    P =   -0.076 deg,    R =   -0.996 deg
};
P[176]{
   GP1:
    UF : 0, UT : 6,      CONFIG : 'N U T, 0, 0, 0',
    X =  418.035  mm,    Y =   -55.273  mm,    Z =   679.797  mm,
    W =  -175.901 deg,    P =   -0.071 deg,    R =   -0.997 deg
};
P[177]{
   GP1:
    UF : 0, UT : 6,      CONFIG : 'N U T, 0, 0, 0',
    X =  418.229  mm,    Y =   -59.852  mm,    Z =   681.326  mm,
    W =  -176.732 deg,    P =   -0.057 deg,    R =   -0.997 deg
};
P[178]{
   GP1:
    UF : 0, UT : 6,      CONFIG : 'N U T, 0, 0, 0',
    X =  418.016  mm,    Y =   -75.862  mm,    Z =   702.954  mm,
    W =  -180.022 deg,    P =   0.000 deg,    R =   -0.999 deg
};
P[179]{
   GP1:
    UF : 0, UT : 6,      CONFIG : 'N U T, 0, 0, 0',
    X =  418.294  mm,    Y =   -81.243  mm,    Z =   700.152  mm,
    W =  -181.016 deg,    P =   0.018 deg,    R =   -0.999 deg
};
P[180]{
   GP1:
    UF : 0, UT : 6,      CONFIG : 'N U T, 0, 0, 0',
    X =  417.953  mm,    Y =   -87.551  mm,    Z =   694.540  mm,
    W =  -182.730 deg,    P =   0.048 deg,    R =   -0.998 deg
};
P[181]{
   GP1:
    UF : 0, UT : 6,      CONFIG : 'N U T, 0, 0, 0',
    X =  418.614  mm,    Y =   -96.970  mm,    Z =   685.674  mm,
    W =  -185.462 deg,    P =   0.095 deg,    R =   -0.995 deg
};
P[182]{
   GP1:
    UF : 0, UT : 6,      CONFIG : 'N U T, 0, 0, 0',
    X =  418.524  mm,    Y =   -101.517  mm,    Z =   673.223  mm,
    W =  -187.120 deg,    P =   0.124 deg,    R =   -0.992 deg
};
P[183]{
   GP1:
    UF : 0, UT : 6,      CONFIG : 'N U T, 0, 0, 0',
    X =  419.264  mm,    Y =   -106.365  mm,    Z =   673.223  mm,
    W =  -188.785 deg,    P =   0.153 deg,    R =   -0.988 deg
};
P[184]{
   GP1:
    UF : 0, UT : 6,      CONFIG : 'N U T, 0, 0, 0',
    X =  417.921  mm,    Y =   -110.829  mm,    Z =   673.223  mm,
    W =  -190.769 deg,    P =   0.187 deg,    R =   -0.982 deg
};
P[185]{
   GP1:
    UF : 0, UT : 6,      CONFIG : 'N U T, 0, 0, 0',
    X =  420.000  mm,    Y =   -206.397  mm,    Z =   673.223  mm,
    W =  -180.000 deg,    P =   0.000 deg,    R =   0.000 deg
};
P[186]{
   GP1:
    UF : 0, UT : 6,      CONFIG : 'N U T, 0, 0, 0',
    X =  383.647  mm,    Y =   -206.397  mm,    Z =   674.929  mm,
    W =  -180.000 deg,    P =   0.000 deg,    R =   0.000 deg
};
P[187]{
   GP1:
    UF : 0, UT : 6,      CONFIG : 'N U T, 0, 0, 0',
    X =  382.227  mm,    Y =   -121.494  mm,    Z =   674.929  mm,
    W =  -192.262 deg,    P =   0.212 deg,    R =   -0.977 deg
};
P[188]{
   GP1:
    UF : 0, UT : 6,      CONFIG : 'N U T, 0, 0, 0',
    X =  382.665  mm,    Y =   -116.759  mm,    Z =   674.929  mm,
    W =  -191.346 deg,    P =   0.197 deg,    R =   -0.980 deg
};
P[189]{
   GP1:
    UF : 0, UT : 6,      CONFIG : 'N U T, 0, 0, 0',
    X =  382.691  mm,    Y =   -111.958  mm,    Z =   674.929  mm,
    W =  -190.241 deg,    P =   0.178 deg,    R =   -0.984 deg
};
P[190]{
   GP1:
    UF : 0, UT : 6,      CONFIG : 'N U T, 0, 0, 0',
    X =  382.715  mm,    Y =   -107.370  mm,    Z =   687.240  mm,
    W =  -188.612 deg,    P =   0.150 deg,    R =   -0.989 deg
};
P[191]{
   GP1:
    UF : 0, UT : 6,      CONFIG : 'N U T, 0, 0, 0',
    X =  382.739  mm,    Y =   -102.993  mm,    Z =   690.953  mm,
    W =  -187.317 deg,    P =   0.127 deg,    R =   -0.992 deg
};
P[192]{
   GP1:
    UF : 0, UT : 6,      CONFIG : 'N U T, 0, 0, 0',
    X =  382.762  mm,    Y =   -98.457  mm,    Z =   694.959  mm,
    W =  -185.995 deg,    P =   0.104 deg,    R =   -0.994 deg
};
P[193]{
   GP1:
    UF : 0, UT : 6,      CONFIG : 'N U T, 0, 0, 0',
    X =  382.784  mm,    Y =   -94.313  mm,    Z =   698.418  mm,
    W =  -185.077 deg,    P =   0.088 deg,    R =   -0.996 deg
};
P[194]{
   GP1:
    UF : 0, UT : 6,      CONFIG : 'N U T, 0, 0, 0',
    X =  382.798  mm,    Y =   -89.736  mm,    Z =   699.760  mm,
    W =  -183.633 deg,    P =   0.063 deg,    R =   -0.998 deg
};
P[195]{
   GP1:
    UF : 0, UT : 6,      CONFIG : 'N U T, 0, 0, 0',
    X =  382.499  mm,    Y =   -85.109  mm,    Z =   700.094  mm,
    W =  -182.294 deg,    P =   0.040 deg,    R =   -0.999 deg
};
P[196]{
   GP1:
    UF : 0, UT : 6,      CONFIG : 'N U T, 0, 0, 0',
    X =  383.202  mm,    Y =   -82.352  mm,    Z =   700.553  mm,
    W =  -181.500 deg,    P =   0.026 deg,    R =   -0.999 deg
};
P[197]{
   GP1:
    UF : 0, UT : 6,      CONFIG : 'N U T, 0, 0, 0',
    X =  382.060  mm,    Y =   -76.248  mm,    Z =   700.170  mm,
    W =  -179.948 deg,    P =   -0.001 deg,    R =   -0.999 deg
};
P[198]{
   GP1:
    UF : 0, UT : 6,      CONFIG : 'N U T, 0, 0, 0',
    X =  382.723  mm,    Y =   -72.549  mm,    Z =   697.164  mm,
    W =  -178.983 deg,    P =   -0.018 deg,    R =   -0.999 deg
};
P[199]{
   GP1:
    UF : 0, UT : 6,      CONFIG : 'N U T, 0, 0, 0',
    X =  382.682  mm,    Y =   -67.414  mm,    Z =   698.258  mm,
    W =  -177.935 deg,    P =   -0.036 deg,    R =   -0.998 deg
};
P[200]{
   GP1:
    UF : 0, UT : 6,      CONFIG : 'N U T, 0, 0, 0',
    X =  383.650  mm,    Y =   -62.199  mm,    Z =   698.935  mm,
    W =  -176.999 deg,    P =   -0.052 deg,    R =   -0.998 deg
};
P[201]{
   GP1:
    UF : 0, UT : 6,      CONFIG : 'N U T, 0, 0, 0',
    X =  382.901  mm,    Y =   -56.187  mm,    Z =   698.668  mm,
    W =  -176.089 deg,    P =   -0.068 deg,    R =   -0.997 deg
};
P[202]{
   GP1:
    UF : 0, UT : 6,      CONFIG : 'N U T, 0, 0, 0',
    X =  383.061  mm,    Y =   -50.333  mm,    Z =   698.153  mm,
    W =  -175.137 deg,    P =   -0.085 deg,    R =   -0.995 deg
};
P[203]{
   GP1:
    UF : 0, UT : 6,      CONFIG : 'N U T, 0, 0, 0',
    X =  382.469  mm,    Y =   -45.757  mm,    Z =   697.768  mm,
    W =  -174.625 deg,    P =   -0.094 deg,    R =   -0.995 deg
};
P[204]{
   GP1:
    UF : 0, UT : 6,      CONFIG : 'N U T, 0, 0, 0',
    X =  382.946  mm,    Y =   -41.040  mm,    Z =   697.558  mm,
    W =  -174.088 deg,    P =   -0.103 deg,    R =   -0.994 deg
};
P[205]{
   GP1:
    UF : 0, UT : 6,      CONFIG : 'N U T, 0, 0, 0',
    X =  382.974  mm,    Y =   -35.645  mm,    Z =   697.878  mm,
    W =  -173.558 deg,    P =   -0.112 deg,    R =   -0.993 deg
};
P[206]{
   GP1:
    UF : 0, UT : 6,      CONFIG : 'N U T, 0, 0, 0',
    X =  383.044  mm,    Y =   -32.462  mm,    Z =   697.103  mm,
    W =  -173.269 deg,    P =   -0.117 deg,    R =   -0.992 deg
};
P[207]{
   GP1:
    UF : 0, UT : 6,      CONFIG : 'N U T, 0, 0, 0',
    X =  383.231  mm,    Y =   -27.764  mm,    Z =   697.192  mm,
    W =  -172.802 deg,    P =   -0.125 deg,    R =   -0.991 deg
};
P[208]{
   GP1:
    UF : 0, UT : 6,      CONFIG : 'N U T, 0, 0, 0',
    X =  382.834  mm,    Y =   -21.671  mm,    Z =   696.531  mm,
    W =  -172.065 deg,    P =   -0.138 deg,    R =   -0.990 deg
};
P[209]{
   GP1:
    UF : 0, UT : 6,      CONFIG : 'N U T, 0, 0, 0',
    X =  383.028  mm,    Y =   -15.950  mm,    Z =   693.910  mm,
    W =  -171.301 deg,    P =   -0.151 deg,    R =   -0.988 deg
};
P[210]{
   GP1:
    UF : 0, UT : 6,      CONFIG : 'N U T, 0, 0, 0',
    X =  383.348  mm,    Y =   -12.160  mm,    Z =   691.394  mm,
    W =  -170.796 deg,    P =   -0.160 deg,    R =   -0.986 deg
};
P[211]{
   GP1:
    UF : 0, UT : 6,      CONFIG : 'N U T, 0, 0, 0',
    X =  382.897  mm,    Y =   -8.352  mm,    Z =   688.889  mm,
    W =  -170.512 deg,    P =   -0.165 deg,    R =   -0.986 deg
};
P[212]{
   GP1:
    UF : 0, UT : 6,      CONFIG : 'N U T, 0, 0, 0',
    X =  382.370  mm,    Y =   -4.118  mm,    Z =   685.855  mm,
    W =  -170.294 deg,    P =   -0.168 deg,    R =   -0.985 deg
};
P[213]{
   GP1:
    UF : 0, UT : 6,      CONFIG : 'N U T, 0, 0, 0',
    X =  383.504  mm,    Y =   -0.271  mm,    Z =   683.370  mm,
    W =  -170.232 deg,    P =   -0.170 deg,    R =   -0.985 deg
};
P[214]{
   GP1:
    UF : 0, UT : 6,      CONFIG : 'N U T, 0, 0, 0',
    X =  383.064  mm,    Y =   3.593  mm,    Z =   680.895  mm,
    W =  -170.180 deg,    P =   -0.170 deg,    R =   -0.985 deg
};
P[215]{
   GP1:
    UF : 0, UT : 6,      CONFIG : 'N U T, 0, 0, 0',
    X =  383.229  mm,    Y =   9.323  mm,    Z =   677.335  mm,
    W =  -170.430 deg,    P =   -0.166 deg,    R =   -0.986 deg
};
P[216]{
   GP1:
    UF : 0, UT : 6,      CONFIG : 'N U T, 0, 0, 0',
    X =  382.763  mm,    Y =   13.254  mm,    Z =   675.784  mm,
    W =  -170.772 deg,    P =   -0.160 deg,    R =   -0.987 deg
};
P[217]{
   GP1:
    UF : 0, UT : 6,      CONFIG : 'N U T, 0, 0, 0',
    X =  383.287  mm,    Y =   19.592  mm,    Z =   675.999  mm,
    W =  -171.280 deg,    P =   -0.152 deg,    R =   -0.988 deg
};
P[218]{
   GP1:
    UF : 0, UT : 6,      CONFIG : 'N U T, 0, 0, 0',
    X =  383.118  mm,    Y =   24.680  mm,    Z =   675.873  mm,
    W =  -171.669 deg,    P =   -0.145 deg,    R =   -0.989 deg
};
P[219]{
   GP1:
    UF : 0, UT : 6,      CONFIG : 'N U T, 0, 0, 0',
    X =  382.904  mm,    Y =   28.121  mm,    Z =   675.437  mm,
    W =  -171.951 deg,    P =   -0.140 deg,    R =   -0.990 deg
};
P[220]{
   GP1:
    UF : 0, UT : 6,      CONFIG : 'N U T, 0, 0, 0',
    X =  382.528  mm,    Y =   33.997  mm,    Z =   674.598  mm,
    W =  -172.210 deg,    P =   -0.136 deg,    R =   -0.991 deg
};
P[221]{
   GP1:
    UF : 0, UT : 6,      CONFIG : 'N U T, 0, 0, 0',
    X =  382.259  mm,    Y =   39.256  mm,    Z =   674.563  mm,
    W =  -172.496 deg,    P =   -0.131 deg,    R =   -0.991 deg
};
P[222]{
   GP1:
    UF : 0, UT : 6,      CONFIG : 'N U T, 0, 0, 0',
    X =  382.927  mm,    Y =   42.428  mm,    Z =   674.551  mm,
    W =  -172.696 deg,    P =   -0.127 deg,    R =   -0.992 deg
};
P[223]{
   GP1:
    UF : 0, UT : 6,      CONFIG : 'N U T, 0, 0, 0',
    X =  383.493  mm,    Y =   47.737  mm,    Z =   674.542  mm,
    W =  -173.183 deg,    P =   -0.119 deg,    R =   -0.993 deg
};
P[224]{
   GP1:
    UF : 0, UT : 6,      CONFIG : 'N U T, 0, 0, 0',
    X =  383.197  mm,    Y =   53.296  mm,    Z =   674.289  mm,
    W =  -173.690 deg,    P =   -0.110 deg,    R =   -0.994 deg
};
P[225]{
   GP1:
    UF : 0, UT : 6,      CONFIG : 'N U T, 0, 0, 0',
    X =  382.969  mm,    Y =   56.959  mm,    Z =   673.782  mm,
    W =  -174.142 deg,    P =   -0.102 deg,    R =   -0.995 deg
};
P[226]{
   GP1:
    UF : 0, UT : 6,      CONFIG : 'N U T, 0, 0, 0',
    X =  383.324  mm,    Y =   76.307  mm,    Z =   673.197  mm,
    W =  -176.946 deg,    P =   -0.053 deg,    R =   -0.999 deg
};
P[227]{
   GP1:
    UF : 0, UT : 6,      CONFIG : 'N U T, 0, 0, 0',
    X =  383.521  mm,    Y =   79.982  mm,    Z =   673.566  mm,
    W =  -177.394 deg,    P =   -0.045 deg,    R =   -0.999 deg
};
P[228]{
   GP1:
    UF : 0, UT : 6,      CONFIG : 'N U T, 0, 0, 0',
    X =  383.393  mm,    Y =   82.885  mm,    Z =   673.694  mm,
    W =  -177.817 deg,    P =   -0.038 deg,    R =   -0.999 deg
};
P[229]{
   GP1:
    UF : 0, UT : 6,      CONFIG : 'N U T, 0, 0, 0',
    X =  383.135  mm,    Y =   88.055  mm,    Z =   673.579  mm,
    W =  -178.649 deg,    P =   -0.024 deg,    R =   -1.000 deg
};
P[230]{
   GP1:
    UF : 0, UT : 6,      CONFIG : 'N U T, 0, 0, 0',
    X =  382.925  mm,    Y =   93.295  mm,    Z =   674.038  mm,
    W =  -179.243 deg,    P =   -0.013 deg,    R =   -1.000 deg
};
P[231]{
   GP1:
    UF : 0, UT : 6,      CONFIG : 'N U T, 0, 0, 0',
    X =  382.726  mm,    Y =   98.480  mm,    Z =   674.592  mm,
    W =  -179.874 deg,    P =   -0.002 deg,    R =   -1.000 deg
};
P[232]{
   GP1:
    UF : 0, UT : 6,      CONFIG : 'N U T, 0, 0, 0',
    X =  382.074  mm,    Y =   104.972  mm,    Z =   675.622  mm,
    W =  -180.460 deg,    P =   0.008 deg,    R =   -1.000 deg
};
P[233]{
   GP1:
    UF : 0, UT : 6,      CONFIG : 'N U T, 0, 0, 0',
    X =  382.527  mm,    Y =   109.699  mm,    Z =   675.614  mm,
    W =  -180.639 deg,    P =   0.011 deg,    R =   -1.000 deg
};
P[234]{
   GP1:
    UF : 0, UT : 6,      CONFIG : 'N U T, 0, 0, 0',
    X =  382.859  mm,    Y =   114.411  mm,    Z =   674.883  mm,
    W =  -180.653 deg,    P =   0.011 deg,    R =   -1.000 deg
};
P[235]{
   GP1:
    UF : 0, UT : 6,      CONFIG : 'N U T, 0, 0, 0',
    X =  383.414  mm,    Y =   118.688  mm,    Z =   675.242  mm,
    W =  -180.623 deg,    P =   0.011 deg,    R =   -1.000 deg
};
P[236]{
   GP1:
    UF : 0, UT : 6,      CONFIG : 'N U T, 0, 0, 0',
    X =  383.282  mm,    Y =   124.671  mm,    Z =   675.242  mm,
    W =  -180.648 deg,    P =   0.011 deg,    R =   -1.000 deg
};
P[237]{
   GP1:
    UF : 0, UT : 6,      CONFIG : 'N U T, 0, 0, 0',
    X =  383.647  mm,    Y =   206.397  mm,    Z =   675.242  mm,
    W =  -180.000 deg,    P =   0.000 deg,    R =   0.000 deg
};
P[238]{
   GP1:
    UF : 0, UT : 6,      CONFIG : 'N U T, 0, 0, 0',
    X =  347.294  mm,    Y =   206.397  mm,    Z =   674.706  mm,
    W =  -180.000 deg,    P =   0.000 deg,    R =   0.000 deg
};
P[239]{
   GP1:
    UF : 0, UT : 6,      CONFIG : 'N U T, 0, 0, 0',
    X =  348.131  mm,    Y =   124.018  mm,    Z =   674.706  mm,
    W =  -180.872 deg,    P =   0.015 deg,    R =   -1.000 deg
};
P[240]{
   GP1:
    UF : 0, UT : 6,      CONFIG : 'N U T, 0, 0, 0',
    X =  348.157  mm,    Y =   120.034  mm,    Z =   674.706  mm,
    W =  -180.844 deg,    P =   0.015 deg,    R =   -1.000 deg
};
P[241]{
   GP1:
    UF : 0, UT : 6,      CONFIG : 'N U T, 0, 0, 0',
    X =  347.303  mm,    Y =   114.208  mm,    Z =   676.285  mm,
    W =  -180.808 deg,    P =   0.014 deg,    R =   -1.000 deg
};
P[242]{
   GP1:
    UF : 0, UT : 6,      CONFIG : 'N U T, 0, 0, 0',
    X =  347.791  mm,    Y =   108.835  mm,    Z =   677.015  mm,
    W =  -180.722 deg,    P =   0.013 deg,    R =   -1.000 deg
};
P[243]{
   GP1:
    UF : 0, UT : 6,      CONFIG : 'N U T, 0, 0, 0',
    X =  348.297  mm,    Y =   102.650  mm,    Z =   677.439  mm,
    W =  -180.454 deg,    P =   0.008 deg,    R =   -1.000 deg
};
P[244]{
   GP1:
    UF : 0, UT : 6,      CONFIG : 'N U T, 0, 0, 0',
    X =  348.640  mm,    Y =   97.256  mm,    Z =   677.088  mm,
    W =  -180.071 deg,    P =   0.001 deg,    R =   -1.000 deg
};
P[245]{
   GP1:
    UF : 0, UT : 6,      CONFIG : 'N U T, 0, 0, 0',
    X =  347.489  mm,    Y =   91.681  mm,    Z =   676.671  mm,
    W =  -179.729 deg,    P =   -0.005 deg,    R =   -1.000 deg
};
P[246]{
   GP1:
    UF : 0, UT : 6,      CONFIG : 'N U T, 0, 0, 0',
    X =  347.550  mm,    Y =   87.613  mm,    Z =   676.490  mm,
    W =  -179.232 deg,    P =   -0.013 deg,    R =   -1.000 deg
};
P[247]{
   GP1:
    UF : 0, UT : 6,      CONFIG : 'N U T, 0, 0, 0',
    X =  347.707  mm,    Y =   85.403  mm,    Z =   676.448  mm,
    W =  -178.877 deg,    P =   -0.020 deg,    R =   -1.000 deg
};
P[248]{
   GP1:
    UF : 0, UT : 6,      CONFIG : 'N U T, 0, 0, 0',
    X =  348.169  mm,    Y =   78.843  mm,    Z =   676.295  mm,
    W =  -178.114 deg,    P =   -0.033 deg,    R =   -0.999 deg
};
P[249]{
   GP1:
    UF : 0, UT : 6,      CONFIG : 'N U T, 0, 0, 0',
    X =  348.248  mm,    Y =   73.412  mm,    Z =   676.415  mm,
    W =  -177.508 deg,    P =   -0.043 deg,    R =   -0.999 deg
};
P[250]{
   GP1:
    UF : 0, UT : 6,      CONFIG : 'N U T, 0, 0, 0',
    X =  347.304  mm,    Y =   68.521  mm,    Z =   676.721  mm,
    W =  -176.834 deg,    P =   -0.055 deg,    R =   -0.998 deg
};
P[251]{
   GP1:
    UF : 0, UT : 6,      CONFIG : 'N U T, 0, 0, 0',
    X =  346.882  mm,    Y =   64.125  mm,    Z =   676.602  mm,
    W =  -176.331 deg,    P =   -0.064 deg,    R =   -0.998 deg
};
P[252]{
   GP1:
    UF : 0, UT : 6,      CONFIG : 'N U T, 0, 0, 0',
    X =  348.130  mm,    Y =   57.610  mm,    Z =   676.771  mm,
    W =  -175.437 deg,    P =   -0.080 deg,    R =   -0.997 deg
};
P[253]{
   GP1:
    UF : 0, UT : 6,      CONFIG : 'N U T, 0, 0, 0',
    X =  348.018  mm,    Y =   53.670  mm,    Z =   675.998  mm,
    W =  -175.103 deg,    P =   -0.085 deg,    R =   -0.996 deg
};
P[254]{
   GP1:
    UF : 0, UT : 6,      CONFIG : 'N U T, 0, 0, 0',
    X =  348.662  mm,    Y =   47.297  mm,    Z =   675.063  mm,
    W =  -174.532 deg,    P =   -0.095 deg,    R =   -0.995 deg
};
P[255]{
   GP1:
    UF : 0, UT : 6,      CONFIG : 'N U T, 0, 0, 0',
    X =  347.546  mm,    Y =   42.068  mm,    Z =   674.440  mm,
    W =  -174.203 deg,    P =   -0.101 deg,    R =   -0.995 deg
};
P[256]{
   GP1:
    UF : 0, UT : 6,      CONFIG : 'N U T, 0, 0, 0',
    X =  346.714  mm,    Y =   39.256  mm,    Z =   674.563  mm,
    W =  -174.100 deg,    P =   -0.103 deg,    R =   -0.995 deg
};
P[257]{
   GP1:
    UF : 0, UT : 6,      CONFIG : 'N U T, 0, 0, 0',
    X =  347.800  mm,    Y =   33.956  mm,    Z =   674.374  mm,
    W =  -173.646 deg,    P =   -0.111 deg,    R =   -0.994 deg
};
P[258]{
   GP1:
    UF : 0, UT : 6,      CONFIG : 'N U T, 0, 0, 0',
    X =  349.172  mm,    Y =   28.760  mm,    Z =   674.645  mm,
    W =  -173.177 deg,    P =   -0.119 deg,    R =   -0.993 deg
};
P[259]{
   GP1:
    UF : 0, UT : 6,      CONFIG : 'N U T, 0, 0, 0',
    X =  347.860  mm,    Y =   24.596  mm,    Z =   674.696  mm,
    W =  -172.850 deg,    P =   -0.124 deg,    R =   -0.992 deg
};
P[260]{
   GP1:
    UF : 0, UT : 6,      CONFIG : 'N U T, 0, 0, 0',
    X =  347.115  mm,    Y =   19.032  mm,    Z =   675.041  mm,
    W =  -172.403 deg,    P =   -0.132 deg,    R =   -0.991 deg
};
P[261]{
   GP1:
    UF : 0, UT : 6,      CONFIG : 'N U T, 0, 0, 0',
    X =  348.031  mm,    Y =   14.113  mm,    Z =   675.917  mm,
    W =  -172.078 deg,    P =   -0.138 deg,    R =   -0.990 deg
};
P[262]{
   GP1:
    UF : 0, UT : 6,      CONFIG : 'N U T, 0, 0, 0',
    X =  348.386  mm,    Y =   9.579  mm,    Z =   677.329  mm,
    W =  -171.896 deg,    P =   -0.141 deg,    R =   -0.989 deg
};
P[263]{
   GP1:
    UF : 0, UT : 6,      CONFIG : 'N U T, 0, 0, 0',
    X =  347.749  mm,    Y =   4.415  mm,    Z =   679.821  mm,
    W =  -171.658 deg,    P =   -0.145 deg,    R =   -0.988 deg
};
P[264]{
   GP1:
    UF : 0, UT : 6,      CONFIG : 'N U T, 0, 0, 0',
    X =  346.662  mm,    Y =   1.161  mm,    Z =   681.489  mm,
    W =  -171.522 deg,    P =   -0.147 deg,    R =   -0.988 deg
};
P[265]{
   GP1:
    UF : 0, UT : 6,      CONFIG : 'N U T, 0, 0, 0',
    X =  348.007  mm,    Y =   -1.532  mm,    Z =   683.738  mm,
    W =  -171.388 deg,    P =   -0.150 deg,    R =   -0.987 deg
};
P[266]{
   GP1:
    UF : 0, UT : 6,      CONFIG : 'N U T, 0, 0, 0',
    X =  347.968  mm,    Y =   -5.857  mm,    Z =   686.441  mm,
    W =  -171.367 deg,    P =   -0.150 deg,    R =   -0.987 deg
};
P[267]{
   GP1:
    UF : 0, UT : 6,      CONFIG : 'N U T, 0, 0, 0',
    X =  346.927  mm,    Y =   -11.288  mm,    Z =   689.593  mm,
    W =  -171.630 deg,    P =   -0.145 deg,    R =   -0.987 deg
};
P[268]{
   GP1:
    UF : 0, UT : 6,      CONFIG : 'N U T, 0, 0, 0',
    X =  348.779  mm,    Y =   -14.740  mm,    Z =   692.288  mm,
    W =  -171.798 deg,    P =   -0.142 deg,    R =   -0.988 deg
};
P[269]{
   GP1:
    UF : 0, UT : 6,      CONFIG : 'N U T, 0, 0, 0',
    X =  347.668  mm,    Y =   -17.612  mm,    Z =   693.592  mm,
    W =  -172.218 deg,    P =   -0.135 deg,    R =   -0.988 deg
};
P[270]{
   GP1:
    UF : 0, UT : 6,      CONFIG : 'N U T, 0, 0, 0',
    X =  347.217  mm,    Y =   -21.709  mm,    Z =   695.944  mm,
    W =  -172.825 deg,    P =   -0.125 deg,    R =   -0.989 deg
};
P[271]{
   GP1:
    UF : 0, UT : 6,      CONFIG : 'N U T, 0, 0, 0',
    X =  348.337  mm,    Y =   -27.447  mm,    Z =   698.745  mm,
    W =  -173.508 deg,    P =   -0.113 deg,    R =   -0.991 deg
};
P[272]{
   GP1:
    UF : 0, UT : 6,      CONFIG : 'N U T, 0, 0, 0',
    X =  347.983  mm,    Y =   -30.616  mm,    Z =   698.570  mm,
    W =  -174.263 deg,    P =   -0.100 deg,    R =   -0.992 deg
};
P[273]{
   GP1:
    UF : 0, UT : 6,      CONFIG : 'N U T, 0, 0, 0',
    X =  347.722  mm,    Y =   -33.827  mm,    Z =   698.642  mm,
    W =  -174.521 deg,    P =   -0.095 deg,    R =   -0.992 deg
};
P[274]{
   GP1:
    UF : 0, UT : 6,      CONFIG : 'N U T, 0, 0, 0',
    X =  347.682  mm,    Y =   -40.751  mm,    Z =   696.516  mm,
    W =  -174.936 deg,    P =   -0.088 deg,    R =   -0.993 deg
};
P[275]{
   GP1:
    UF : 0, UT : 6,      CONFIG : 'N U T, 0, 0, 0',
    X =  347.820  mm,    Y =   -47.191  mm,    Z =   693.532  mm,
    W =  -175.293 deg,    P =   -0.082 deg,    R =   -0.993 deg
};
P[276]{
   GP1:
    UF : 0, UT : 6,      CONFIG : 'N U T, 0, 0, 0',
    X =  348.116  mm,    Y =   -50.782  mm,    Z =   693.510  mm,
    W =  -175.546 deg,    P =   -0.077 deg,    R =   -0.994 deg
};
P[277]{
   GP1:
    UF : 0, UT : 6,      CONFIG : 'N U T, 0, 0, 0',
    X =  347.795  mm,    Y =   -55.791  mm,    Z =   694.892  mm,
    W =  -175.945 deg,    P =   -0.070 deg,    R =   -0.994 deg
};
P[278]{
   GP1:
    UF : 0, UT : 6,      CONFIG : 'N U T, 0, 0, 0',
    X =  348.000  mm,    Y =   -60.962  mm,    Z =   696.781  mm,
    W =  -176.660 deg,    P =   -0.058 deg,    R =   -0.995 deg
};
P[279]{
   GP1:
    UF : 0, UT : 6,      CONFIG : 'N U T, 0, 0, 0',
    X =  346.948  mm,    Y =   -64.199  mm,    Z =   697.702  mm,
    W =  -177.079 deg,    P =   -0.051 deg,    R =   -0.995 deg
};
P[280]{
   GP1:
    UF : 0, UT : 6,      CONFIG : 'N U T, 0, 0, 0',
    X =  347.915  mm,    Y =   -67.728  mm,    Z =   698.502  mm,
    W =  -177.530 deg,    P =   -0.043 deg,    R =   -0.996 deg
};
P[281]{
   GP1:
    UF : 0, UT : 6,      CONFIG : 'N U T, 0, 0, 0',
    X =  347.407  mm,    Y =   -72.147  mm,    Z =   698.573  mm,
    W =  -178.279 deg,    P =   -0.030 deg,    R =   -0.996 deg
};
P[282]{
   GP1:
    UF : 0, UT : 6,      CONFIG : 'N U T, 0, 0, 0',
    X =  348.001  mm,    Y =   -76.813  mm,    Z =   696.947  mm,
    W =  -178.997 deg,    P =   -0.017 deg,    R =   -0.997 deg
};
P[283]{
   GP1:
    UF : 0, UT : 6,      CONFIG : 'N U T, 0, 0, 0',
    X =  347.654  mm,    Y =   -80.731  mm,    Z =   697.199  mm,
    W =  -179.708 deg,    P =   -0.005 deg,    R =   -0.997 deg
};
P[284]{
   GP1:
    UF : 0, UT : 6,      CONFIG : 'N U T, 0, 0, 0',
    X =  347.834  mm,    Y =   -85.665  mm,    Z =   697.501  mm,
    W =  -180.922 deg,    P =   0.016 deg,    R =   -0.997 deg
};
P[285]{
   GP1:
    UF : 0, UT : 6,      CONFIG : 'N U T, 0, 0, 0',
    X =  349.159  mm,    Y =   -90.374  mm,    Z =   697.527  mm,
    W =  -182.275 deg,    P =   0.040 deg,    R =   -0.997 deg
};
P[286]{
   GP1:
    UF : 0, UT : 6,      CONFIG : 'N U T, 0, 0, 0',
    X =  348.228  mm,    Y =   -95.965  mm,    Z =   695.899  mm,
    W =  -183.414 deg,    P =   0.059 deg,    R =   -0.996 deg
};
P[287]{
   GP1:
    UF : 0, UT : 6,      CONFIG : 'N U T, 0, 0, 0',
    X =  348.052  mm,    Y =   -99.615  mm,    Z =   694.631  mm,
    W =  -184.260 deg,    P =   0.074 deg,    R =   -0.995 deg
};
P[288]{
   GP1:
    UF : 0, UT : 6,      CONFIG : 'N U T, 0, 0, 0',
    X =  347.796  mm,    Y =   -104.026  mm,    Z =   692.257  mm,
    W =  -185.346 deg,    P =   0.093 deg,    R =   -0.994 deg
};
P[289]{
   GP1:
    UF : 0, UT : 6,      CONFIG : 'N U T, 0, 0, 0',
    X =  347.876  mm,    Y =   -108.722  mm,    Z =   688.808  mm,
    W =  -186.827 deg,    P =   0.119 deg,    R =   -0.991 deg
};
P[290]{
   GP1:
    UF : 0, UT : 6,      CONFIG : 'N U T, 0, 0, 0',
    X =  347.243  mm,    Y =   -111.888  mm,    Z =   686.245  mm,
    W =  -187.692 deg,    P =   0.134 deg,    R =   -0.989 deg
};
P[291]{
   GP1:
    UF : 0, UT : 6,      CONFIG : 'N U T, 0, 0, 0',
    X =  348.143  mm,    Y =   -114.529  mm,    Z =   684.251  mm,
    W =  -188.334 deg,    P =   0.145 deg,    R =   -0.988 deg
};
P[292]{
   GP1:
    UF : 0, UT : 6,      CONFIG : 'N U T, 0, 0, 0',
    X =  347.977  mm,    Y =   -118.908  mm,    Z =   675.208  mm,
    W =  -189.584 deg,    P =   0.166 deg,    R =   -0.985 deg
};
P[293]{
   GP1:
    UF : 0, UT : 6,      CONFIG : 'N U T, 0, 0, 0',
    X =  348.298  mm,    Y =   -126.277  mm,    Z =   675.208  mm,
    W =  -191.721 deg,    P =   0.203 deg,    R =   -0.978 deg
};
P[294]{
   GP1:
    UF : 0, UT : 6,      CONFIG : 'N U T, 0, 0, 0',
    X =  347.294  mm,    Y =   -206.397  mm,    Z =   675.208  mm,
    W =  -180.000 deg,    P =   0.000 deg,    R =   0.000 deg
};
P[295]{
   GP1:
    UF : 0, UT : 6,      CONFIG : 'N U T, 0, 0, 0',
    X =  310.941  mm,    Y =   -206.397  mm,    Z =   677.138  mm,
    W =  -180.000 deg,    P =   0.000 deg,    R =   0.000 deg
};
P[296]{
   GP1:
    UF : 0, UT : 6,      CONFIG : 'N U T, 0, 0, 0',
    X =  310.598  mm,    Y =   -116.062  mm,    Z =   677.138  mm,
    W =  -187.328 deg,    P =   0.126 deg,    R =   -0.981 deg
};
P[297]{
   GP1:
    UF : 0, UT : 6,      CONFIG : 'N U T, 0, 0, 0',
    X =  312.548  mm,    Y =   -114.091  mm,    Z =   677.138  mm,
    W =  -186.573 deg,    P =   0.113 deg,    R =   -0.983 deg
};
P[298]{
   GP1:
    UF : 0, UT : 6,      CONFIG : 'N U T, 0, 0, 0',
    X =  313.129  mm,    Y =   -109.868  mm,    Z =   677.138  mm,
    W =  -185.339 deg,    P =   0.092 deg,    R =   -0.985 deg
};
P[299]{
   GP1:
    UF : 0, UT : 6,      CONFIG : 'N U T, 0, 0, 0',
    X =  313.115  mm,    Y =   -105.945  mm,    Z =   685.538  mm,
    W =  -184.613 deg,    P =   0.080 deg,    R =   -0.986 deg
};
P[300]{
   GP1:
    UF : 0, UT : 6,      CONFIG : 'N U T, 0, 0, 0',
    X =  312.994  mm,    Y =   -95.602  mm,    Z =   692.874  mm,
    W =  -182.066 deg,    P =   0.036 deg,    R =   -0.989 deg
};
P[301]{
   GP1:
    UF : 0, UT : 6,      CONFIG : 'N U T, 0, 0, 0',
    X =  308.975  mm,    Y =   -91.806  mm,    Z =   693.688  mm,
    W =  -181.350 deg,    P =   0.023 deg,    R =   -0.989 deg
};
P[302]{
   GP1:
    UF : 0, UT : 6,      CONFIG : 'N U T, 0, 0, 0',
    X =  312.566  mm,    Y =   -85.650  mm,    Z =   694.630  mm,
    W =  -180.302 deg,    P =   0.005 deg,    R =   -0.990 deg
};
P[303]{
   GP1:
    UF : 0, UT : 6,      CONFIG : 'N U T, 0, 0, 0',
    X =  312.722  mm,    Y =   -81.526  mm,    Z =   693.884  mm,
    W =  -179.501 deg,    P =   -0.009 deg,    R =   -0.991 deg
};
P[304]{
   GP1:
    UF : 0, UT : 6,      CONFIG : 'N U T, 0, 0, 0',
    X =  312.843  mm,    Y =   -77.565  mm,    Z =   692.911  mm,
    W =  -178.939 deg,    P =   -0.018 deg,    R =   -0.991 deg
};
P[305]{
   GP1:
    UF : 0, UT : 6,      CONFIG : 'N U T, 0, 0, 0',
    X =  312.981  mm,    Y =   -70.524  mm,    Z =   693.961  mm,
    W =  -178.024 deg,    P =   -0.034 deg,    R =   -0.991 deg
};
P[306]{
   GP1:
    UF : 0, UT : 6,      CONFIG : 'N U T, 0, 0, 0',
    X =  312.916  mm,    Y =   -65.151  mm,    Z =   694.004  mm,
    W =  -177.265 deg,    P =   -0.047 deg,    R =   -0.991 deg
};
P[307]{
   GP1:
    UF : 0, UT : 6,      CONFIG : 'N U T, 0, 0, 0',
    X =  313.092  mm,    Y =   -59.599  mm,    Z =   693.353  mm,
    W =  -176.698 deg,    P =   -0.057 deg,    R =   -0.991 deg
};
P[308]{
   GP1:
    UF : 0, UT : 6,      CONFIG : 'N U T, 0, 0, 0',
    X =  312.902  mm,    Y =   -54.791  mm,    Z =   692.997  mm,
    W =  -176.155 deg,    P =   -0.067 deg,    R =   -0.991 deg
};
P[309]{
   GP1:
    UF : 0, UT : 6,      CONFIG : 'N U T, 0, 0, 0',
    X =  313.100  mm,    Y =   -51.298  mm,    Z =   692.750  mm,
    W =  -175.845 deg,    P =   -0.072 deg,    R =   -0.990 deg
};
P[310]{
   GP1:
    UF : 0, UT : 6,      CONFIG : 'N U T, 0, 0, 0',
    X =  313.048  mm,    Y =   -46.750  mm,    Z =   692.886  mm,
    W =  -175.540 deg,    P =   -0.077 deg,    R =   -0.990 deg
};
P[311]{
   GP1:
    UF : 0, UT : 6,      CONFIG : 'N U T, 0, 0, 0',
    X =  312.731  mm,    Y =   -27.076  mm,    Z =   687.144  mm,
    W =  -174.510 deg,    P =   -0.095 deg,    R =   -0.990 deg
};
P[312]{
   GP1:
    UF : 0, UT : 6,      CONFIG : 'N U T, 0, 0, 0',
    X =  313.067  mm,    Y =   -21.254  mm,    Z =   684.294  mm,
    W =  -174.191 deg,    P =   -0.101 deg,    R =   -0.990 deg
};
P[313]{
   GP1:
    UF : 0, UT : 6,      CONFIG : 'N U T, 0, 0, 0',
    X =  312.464  mm,    Y =   -11.460  mm,    Z =   678.742  mm,
    W =  -173.938 deg,    P =   -0.105 deg,    R =   -0.990 deg
};
P[314]{
   GP1:
    UF : 0, UT : 6,      CONFIG : 'N U T, 0, 0, 0',
    X =  313.005  mm,    Y =   -4.970  mm,    Z =   675.802  mm,
    W =  -173.745 deg,    P =   -0.109 deg,    R =   -0.991 deg
};
P[315]{
   GP1:
    UF : 0, UT : 6,      CONFIG : 'N U T, 0, 0, 0',
    X =  311.332  mm,    Y =   -1.432  mm,    Z =   674.447  mm,
    W =  -173.949 deg,    P =   -0.105 deg,    R =   -0.992 deg
};
P[316]{
   GP1:
    UF : 0, UT : 6,      CONFIG : 'N U T, 0, 0, 0',
    X =  312.641  mm,    Y =   8.684  mm,    Z =   674.447  mm,
    W =  -174.182 deg,    P =   -0.101 deg,    R =   -0.993 deg
};
P[317]{
   GP1:
    UF : 0, UT : 6,      CONFIG : 'N U T, 0, 0, 0',
    X =  313.031  mm,    Y =   13.441  mm,    Z =   674.616  mm,
    W =  -174.375 deg,    P =   -0.098 deg,    R =   -0.994 deg
};
P[318]{
   GP1:
    UF : 0, UT : 6,      CONFIG : 'N U T, 0, 0, 0',
    X =  312.609  mm,    Y =   24.878  mm,    Z =   674.343  mm,
    W =  -175.131 deg,    P =   -0.085 deg,    R =   -0.996 deg
};
P[319]{
   GP1:
    UF : 0, UT : 6,      CONFIG : 'N U T, 0, 0, 0',
    X =  313.123  mm,    Y =   31.413  mm,    Z =   673.677  mm,
    W =  -175.673 deg,    P =   -0.075 deg,    R =   -0.997 deg
};
P[320]{
   GP1:
    UF : 0, UT : 6,      CONFIG : 'N U T, 0, 0, 0',
    X =  313.039  mm,    Y =   36.419  mm,    Z =   674.187  mm,
    W =  -176.002 deg,    P =   -0.070 deg,    R =   -0.997 deg
};
P[321]{
   GP1:
    UF : 0, UT : 6,      CONFIG : 'N U T, 0, 0, 0',
    X =  312.344  mm,    Y =   41.716  mm,    Z =   674.455  mm,
    W =  -176.336 deg,    P =   -0.064 deg,    R =   -0.998 deg
};
P[322]{
   GP1:
    UF : 0, UT : 6,      CONFIG : 'N U T, 0, 0, 0',
    X =  312.244  mm,    Y =   46.856  mm,    Z =   675.584  mm,
    W =  -176.700 deg,    P =   -0.058 deg,    R =   -0.998 deg
};
P[323]{
   GP1:
    UF : 0, UT : 6,      CONFIG : 'N U T, 0, 0, 0',
    X =  313.117  mm,    Y =   58.122  mm,    Z =   677.421  mm,
    W =  -177.516 deg,    P =   -0.043 deg,    R =   -0.999 deg
};
P[324]{
   GP1:
    UF : 0, UT : 6,      CONFIG : 'N U T, 0, 0, 0',
    X =  312.689  mm,    Y =   62.430  mm,    Z =   677.446  mm,
    W =  -178.066 deg,    P =   -0.034 deg,    R =   -0.999 deg
};
P[325]{
   GP1:
    UF : 0, UT : 6,      CONFIG : 'N U T, 0, 0, 0',
    X =  312.853  mm,    Y =   68.293  mm,    Z =   676.977  mm,
    W =  -178.675 deg,    P =   -0.023 deg,    R =   -1.000 deg
};
P[326]{
   GP1:
    UF : 0, UT : 6,      CONFIG : 'N U T, 0, 0, 0',
    X =  313.058  mm,    Y =   73.332  mm,    Z =   676.259  mm,
    W =  -179.083 deg,    P =   -0.016 deg,    R =   -1.000 deg
};
P[327]{
   GP1:
    UF : 0, UT : 6,      CONFIG : 'N U T, 0, 0, 0',
    X =  312.476  mm,    Y =   78.603  mm,    Z =   675.947  mm,
    W =  -179.661 deg,    P =   -0.006 deg,    R =   -1.000 deg
};
P[328]{
   GP1:
    UF : 0, UT : 6,      CONFIG : 'N U T, 0, 0, 0',
    X =  312.622  mm,    Y =   93.606  mm,    Z =   675.525  mm,
    W =  -180.596 deg,    P =   0.010 deg,    R =   -1.000 deg
};
P[329]{
   GP1:
    UF : 0, UT : 6,      CONFIG : 'N U T, 0, 0, 0',
    X =  312.239  mm,    Y =   98.328  mm,    Z =   675.959  mm,
    W =  -180.734 deg,    P =   0.013 deg,    R =   -1.000 deg
};
P[330]{
   GP1:
    UF : 0, UT : 6,      CONFIG : 'N U T, 0, 0, 0',
    X =  313.072  mm,    Y =   108.028  mm,    Z =   676.473  mm,
    W =  -180.878 deg,    P =   0.015 deg,    R =   -1.000 deg
};
P[331]{
   GP1:
    UF : 0, UT : 6,      CONFIG : 'N U T, 0, 0, 0',
    X =  312.516  mm,    Y =   114.086  mm,    Z =   676.687  mm,
    W =  -180.939 deg,    P =   0.016 deg,    R =   -1.000 deg
};
P[332]{
   GP1:
    UF : 0, UT : 6,      CONFIG : 'N U T, 0, 0, 0',
    X =  312.522  mm,    Y =   119.507  mm,    Z =   676.687  mm,
    W =  -180.960 deg,    P =   0.017 deg,    R =   -1.000 deg
};
P[333]{
   GP1:
    UF : 0, UT : 6,      CONFIG : 'N U T, 0, 0, 0',
    X =  310.941  mm,    Y =   206.397  mm,    Z =   676.687  mm,
    W =  -180.000 deg,    P =   0.000 deg,    R =   0.000 deg
};
P[334]{
   GP1:
    UF : 0, UT : 6,      CONFIG : 'N U T, 0, 0, 0',
    X =  274.589  mm,    Y =   206.397  mm,    Z =   679.040  mm,
    W =  -180.000 deg,    P =   0.000 deg,    R =   0.000 deg
};
P[335]{
   GP1:
    UF : 0, UT : 6,      CONFIG : 'N U T, 0, 0, 0',
    X =  273.192  mm,    Y =   123.826  mm,    Z =   679.040  mm,
    W =  -180.903 deg,    P =   0.016 deg,    R =   -1.000 deg
};
P[336]{
   GP1:
    UF : 0, UT : 6,      CONFIG : 'N U T, 0, 0, 0',
    X =  272.696  mm,    Y =   118.912  mm,    Z =   679.040  mm,
    W =  -180.942 deg,    P =   0.016 deg,    R =   -1.000 deg
};
P[337]{
   GP1:
    UF : 0, UT : 6,      CONFIG : 'N U T, 0, 0, 0',
    X =  272.480  mm,    Y =   114.824  mm,    Z =   679.040  mm,
    W =  -180.965 deg,    P =   0.017 deg,    R =   -1.000 deg
};
P[338]{
   GP1:
    UF : 0, UT : 6,      CONFIG : 'N U T, 0, 0, 0',
    X =  273.847  mm,    Y =   111.147  mm,    Z =   678.811  mm,
    W =  -180.991 deg,    P =   0.017 deg,    R =   -1.000 deg
};
P[339]{
   GP1:
    UF : 0, UT : 6,      CONFIG : 'N U T, 0, 0, 0',
    X =  272.816  mm,    Y =   107.746  mm,    Z =   678.135  mm,
    W =  -181.015 deg,    P =   0.018 deg,    R =   -1.000 deg
};
P[340]{
   GP1:
    UF : 0, UT : 6,      CONFIG : 'N U T, 0, 0, 0',
    X =  272.520  mm,    Y =   102.411  mm,    Z =   677.689  mm,
    W =  -181.039 deg,    P =   0.018 deg,    R =   -1.000 deg
};
P[341]{
   GP1:
    UF : 0, UT : 6,      CONFIG : 'N U T, 0, 0, 0',
    X =  273.073  mm,    Y =   97.137  mm,    Z =   677.213  mm,
    W =  -181.072 deg,    P =   0.019 deg,    R =   -1.000 deg
};
P[342]{
   GP1:
    UF : 0, UT : 6,      CONFIG : 'N U T, 0, 0, 0',
    X =  272.997  mm,    Y =   92.047  mm,    Z =   676.583  mm,
    W =  -181.119 deg,    P =   0.020 deg,    R =   -1.000 deg
};
P[343]{
   GP1:
    UF : 0, UT : 6,      CONFIG : 'N U T, 0, 0, 0',
    X =  272.397  mm,    Y =   87.613  mm,    Z =   676.490  mm,
    W =  -181.124 deg,    P =   0.020 deg,    R =   -1.000 deg
};
P[344]{
   GP1:
    UF : 0, UT : 6,      CONFIG : 'N U T, 0, 0, 0',
    X =  272.669  mm,    Y =   85.403  mm,    Z =   676.448  mm,
    W =  -181.101 deg,    P =   0.019 deg,    R =   -1.000 deg
};
P[345]{
   GP1:
    UF : 0, UT : 6,      CONFIG : 'N U T, 0, 0, 0',
    X =  273.060  mm,    Y =   78.804  mm,    Z =   676.337  mm,
    W =  -181.043 deg,    P =   0.018 deg,    R =   -1.000 deg
};
P[346]{
   GP1:
    UF : 0, UT : 6,      CONFIG : 'N U T, 0, 0, 0',
    X =  273.158  mm,    Y =   70.123  mm,    Z =   677.384  mm,
    W =  -180.794 deg,    P =   0.014 deg,    R =   -1.000 deg
};
P[347]{
   GP1:
    UF : 0, UT : 6,      CONFIG : 'N U T, 0, 0, 0',
    X =  273.007  mm,    Y =   66.183  mm,    Z =   678.121  mm,
    W =  -180.668 deg,    P =   0.012 deg,    R =   -1.000 deg
};
P[348]{
   GP1:
    UF : 0, UT : 6,      CONFIG : 'N U T, 0, 0, 0',
    X =  272.674  mm,    Y =   62.715  mm,    Z =   678.353  mm,
    W =  -180.444 deg,    P =   0.008 deg,    R =   -1.000 deg
};
P[349]{
   GP1:
    UF : 0, UT : 6,      CONFIG : 'N U T, 0, 0, 0',
    X =  273.970  mm,    Y =   59.371  mm,    Z =   678.463  mm,
    W =  -180.159 deg,    P =   0.003 deg,    R =   -1.000 deg
};
P[350]{
   GP1:
    UF : 0, UT : 6,      CONFIG : 'N U T, 0, 0, 0',
    X =  273.293  mm,    Y =   56.515  mm,    Z =   678.562  mm,
    W =  -180.066 deg,    P =   0.001 deg,    R =   -1.000 deg
};
P[351]{
   GP1:
    UF : 0, UT : 6,      CONFIG : 'N U T, 0, 0, 0',
    X =  273.710  mm,    Y =   44.828  mm,    Z =   676.888  mm,
    W =  -179.269 deg,    P =   -0.013 deg,    R =   -1.000 deg
};
P[352]{
   GP1:
    UF : 0, UT : 6,      CONFIG : 'N U T, 0, 0, 0',
    X =  273.113  mm,    Y =   40.491  mm,    Z =   675.927  mm,
    W =  -178.963 deg,    P =   -0.018 deg,    R =   -1.000 deg
};
P[353]{
   GP1:
    UF : 0, UT : 6,      CONFIG : 'N U T, 0, 0, 0',
    X =  272.855  mm,    Y =   33.976  mm,    Z =   675.578  mm,
    W =  -178.550 deg,    P =   -0.025 deg,    R =   -0.999 deg
};
P[354]{
   GP1:
    UF : 0, UT : 6,      CONFIG : 'N U T, 0, 0, 0',
    X =  273.265  mm,    Y =   28.972  mm,    Z =   676.213  mm,
    W =  -178.240 deg,    P =   -0.031 deg,    R =   -0.999 deg
};
P[355]{
   GP1:
    UF : 0, UT : 6,      CONFIG : 'N U T, 0, 0, 0',
    X =  272.857  mm,    Y =   23.581  mm,    Z =   676.610  mm,
    W =  -177.949 deg,    P =   -0.036 deg,    R =   -0.999 deg
};
P[356]{
   GP1:
    UF : 0, UT : 6,      CONFIG : 'N U T, 0, 0, 0',
    X =  273.113  mm,    Y =   18.155  mm,    Z =   676.368  mm,
    W =  -177.569 deg,    P =   -0.042 deg,    R =   -0.998 deg
};
P[357]{
   GP1:
    UF : 0, UT : 6,      CONFIG : 'N U T, 0, 0, 0',
    X =  273.273  mm,    Y =   14.369  mm,    Z =   676.280  mm,
    W =  -177.296 deg,    P =   -0.047 deg,    R =   -0.998 deg
};
P[358]{
   GP1:
    UF : 0, UT : 6,      CONFIG : 'N U T, 0, 0, 0',
    X =  272.543  mm,    Y =   9.437  mm,    Z =   675.885  mm,
    W =  -177.075 deg,    P =   -0.051 deg,    R =   -0.997 deg
};
P[359]{
   GP1:
    UF : 0, UT : 6,      CONFIG : 'N U T, 0, 0, 0',
    X =  273.198  mm,    Y =   2.350  mm,    Z =   674.697  mm,
    W =  -176.653 deg,    P =   -0.058 deg,    R =   -0.996 deg
};
P[360]{
   GP1:
    UF : 0, UT : 6,      CONFIG : 'N U T, 0, 0, 0',
    X =  272.640  mm,    Y =   -3.852  mm,    Z =   674.718  mm,
    W =  -176.468 deg,    P =   -0.061 deg,    R =   -0.995 deg
};
P[361]{
   GP1:
    UF : 0, UT : 6,      CONFIG : 'N U T, 0, 0, 0',
    X =  273.083  mm,    Y =   -11.223  mm,    Z =   674.086  mm,
    W =  -176.292 deg,    P =   -0.064 deg,    R =   -0.994 deg
};
P[362]{
   GP1:
    UF : 0, UT : 6,      CONFIG : 'N U T, 0, 0, 0',
    X =  272.869  mm,    Y =   -15.871  mm,    Z =   674.132  mm,
    W =  -176.222 deg,    P =   -0.066 deg,    R =   -0.994 deg
};
P[363]{
   GP1:
    UF : 0, UT : 6,      CONFIG : 'N U T, 0, 0, 0',
    X =  272.941  mm,    Y =   -20.568  mm,    Z =   673.962  mm,
    W =  -176.232 deg,    P =   -0.065 deg,    R =   -0.993 deg
};
P[364]{
   GP1:
    UF : 0, UT : 6,      CONFIG : 'N U T, 0, 0, 0',
    X =  272.839  mm,    Y =   -26.886  mm,    Z =   675.070  mm,
    W =  -176.237 deg,    P =   -0.065 deg,    R =   -0.992 deg
};
P[365]{
   GP1:
    UF : 0, UT : 6,      CONFIG : 'N U T, 0, 0, 0',
    X =  272.826  mm,    Y =   -33.731  mm,    Z =   675.584  mm,
    W =  -176.301 deg,    P =   -0.064 deg,    R =   -0.992 deg
};
P[366]{
   GP1:
    UF : 0, UT : 6,      CONFIG : 'N U T, 0, 0, 0',
    X =  273.084  mm,    Y =   -40.800  mm,    Z =   676.025  mm,
    W =  -176.349 deg,    P =   -0.063 deg,    R =   -0.991 deg
};
P[367]{
   GP1:
    UF : 0, UT : 6,      CONFIG : 'N U T, 0, 0, 0',
    X =  273.051  mm,    Y =   -45.784  mm,    Z =   676.914  mm,
    W =  -176.531 deg,    P =   -0.060 deg,    R =   -0.991 deg
};
P[368]{
   GP1:
    UF : 0, UT : 6,      CONFIG : 'N U T, 0, 0, 0',
    X =  272.458  mm,    Y =   -52.290  mm,    Z =   678.929  mm,
    W =  -176.937 deg,    P =   -0.053 deg,    R =   -0.990 deg
};
P[369]{
   GP1:
    UF : 0, UT : 6,      CONFIG : 'N U T, 0, 0, 0',
    X =  272.471  mm,    Y =   -60.539  mm,    Z =   680.529  mm,
    W =  -177.409 deg,    P =   -0.045 deg,    R =   -0.989 deg
};
P[370]{
   GP1:
    UF : 0, UT : 6,      CONFIG : 'N U T, 0, 0, 0',
    X =  273.575  mm,    Y =   -65.135  mm,    Z =   681.915  mm,
    W =  -177.763 deg,    P =   -0.039 deg,    R =   -0.989 deg
};
P[371]{
   GP1:
    UF : 0, UT : 6,      CONFIG : 'N U T, 0, 0, 0',
    X =  273.762  mm,    Y =   -71.076  mm,    Z =   682.235  mm,
    W =  -178.230 deg,    P =   -0.031 deg,    R =   -0.989 deg
};
P[372]{
   GP1:
    UF : 0, UT : 6,      CONFIG : 'N U T, 0, 0, 0',
    X =  273.175  mm,    Y =   -76.647  mm,    Z =   681.777  mm,
    W =  -178.531 deg,    P =   -0.025 deg,    R =   -0.988 deg
};
P[373]{
   GP1:
    UF : 0, UT : 6,      CONFIG : 'N U T, 0, 0, 0',
    X =  273.327  mm,    Y =   -80.365  mm,    Z =   680.809  mm,
    W =  -178.905 deg,    P =   -0.019 deg,    R =   -0.988 deg
};
P[374]{
   GP1:
    UF : 0, UT : 6,      CONFIG : 'N U T, 0, 0, 0',
    X =  273.097  mm,    Y =   -83.755  mm,    Z =   679.214  mm,
    W =  -179.176 deg,    P =   -0.014 deg,    R =   -0.988 deg
};
P[375]{
   GP1:
    UF : 0, UT : 6,      CONFIG : 'N U T, 0, 0, 0',
    X =  273.860  mm,    Y =   -90.411  mm,    Z =   677.543  mm,
    W =  -180.004 deg,    P =   0.000 deg,    R =   -0.987 deg
};
P[376]{
   GP1:
    UF : 0, UT : 6,      CONFIG : 'N U T, 0, 0, 0',
    X =  272.713  mm,    Y =   -95.258  mm,    Z =   674.448  mm,
    W =  -180.503 deg,    P =   0.009 deg,    R =   -0.986 deg
};
P[377]{
   GP1:
    UF : 0, UT : 6,      CONFIG : 'N U T, 0, 0, 0',
    X =  275.448  mm,    Y =   -100.353  mm,    Z =   674.448  mm,
    W =  -181.741 deg,    P =   0.030 deg,    R =   -0.985 deg
};
P[378]{
   GP1:
    UF : 0, UT : 6,      CONFIG : 'N U T, 0, 0, 0',
    X =  274.589  mm,    Y =   -206.397  mm,    Z =   674.448  mm,
    W =  -180.000 deg,    P =   0.000 deg,    R =   0.000 deg
};
P[379]{
   GP1:
    UF : 0, UT : 6,      CONFIG : 'N U T, 0, 0, 0',
    X =  238.236  mm,    Y =   -206.397  mm,    Z =   674.531  mm,
    W =  -180.000 deg,    P =   0.000 deg,    R =   0.000 deg
};
P[380]{
   GP1:
    UF : 0, UT : 6,      CONFIG : 'N U T, 0, 0, 0',
    X =  238.008  mm,    Y =   -71.414  mm,    Z =   674.531  mm,
    W =  -178.542 deg,    P =   -0.025 deg,    R =   -0.990 deg
};
P[381]{
   GP1:
    UF : 0, UT : 6,      CONFIG : 'N U T, 0, 0, 0',
    X =  237.934  mm,    Y =   -65.793  mm,    Z =   674.531  mm,
    W =  -178.262 deg,    P =   -0.030 deg,    R =   -0.991 deg
};
P[382]{
   GP1:
    UF : 0, UT : 6,      CONFIG : 'N U T, 0, 0, 0',
    X =  237.826  mm,    Y =   -59.910  mm,    Z =   674.311  mm,
    W =  -177.995 deg,    P =   -0.035 deg,    R =   -0.991 deg
};
P[383]{
   GP1:
    UF : 0, UT : 6,      CONFIG : 'N U T, 0, 0, 0',
    X =  237.534  mm,    Y =   -55.176  mm,    Z =   674.704  mm,
    W =  -177.888 deg,    P =   -0.037 deg,    R =   -0.992 deg
};
P[384]{
   GP1:
    UF : 0, UT : 6,      CONFIG : 'N U T, 0, 0, 0',
    X =  237.884  mm,    Y =   -49.344  mm,    Z =   674.610  mm,
    W =  -177.788 deg,    P =   -0.038 deg,    R =   -0.993 deg
};
P[385]{
   GP1:
    UF : 0, UT : 6,      CONFIG : 'N U T, 0, 0, 0',
    X =  237.084  mm,    Y =   -45.591  mm,    Z =   674.752  mm,
    W =  -177.695 deg,    P =   -0.040 deg,    R =   -0.993 deg
};
P[386]{
   GP1:
    UF : 0, UT : 6,      CONFIG : 'N U T, 0, 0, 0',
    X =  238.399  mm,    Y =   -42.909  mm,    Z =   674.195  mm,
    W =  -177.634 deg,    P =   -0.041 deg,    R =   -0.993 deg
};
P[387]{
   GP1:
    UF : 0, UT : 6,      CONFIG : 'N U T, 0, 0, 0',
    X =  236.880  mm,    Y =   -36.604  mm,    Z =   673.655  mm,
    W =  -177.800 deg,    P =   -0.038 deg,    R =   -0.995 deg
};
P[388]{
   GP1:
    UF : 0, UT : 6,      CONFIG : 'N U T, 0, 0, 0',
    X =  238.410  mm,    Y =   -31.914  mm,    Z =   673.844  mm,
    W =  -177.788 deg,    P =   -0.038 deg,    R =   -0.995 deg
};
P[389]{
   GP1:
    UF : 0, UT : 6,      CONFIG : 'N U T, 0, 0, 0',
    X =  236.674  mm,    Y =   -25.447  mm,    Z =   673.924  mm,
    W =  -178.018 deg,    P =   -0.034 deg,    R =   -0.996 deg
};
P[390]{
   GP1:
    UF : 0, UT : 6,      CONFIG : 'N U T, 0, 0, 0',
    X =  237.896  mm,    Y =   -21.022  mm,    Z =   674.602  mm,
    W =  -178.031 deg,    P =   -0.034 deg,    R =   -0.996 deg
};
P[391]{
   GP1:
    UF : 0, UT : 6,      CONFIG : 'N U T, 0, 0, 0',
    X =  237.567  mm,    Y =   -15.399  mm,    Z =   674.823  mm,
    W =  -178.124 deg,    P =   -0.033 deg,    R =   -0.997 deg
};
P[392]{
   GP1:
    UF : 0, UT : 6,      CONFIG : 'N U T, 0, 0, 0',
    X =  238.149  mm,    Y =   -9.477  mm,    Z =   674.700  mm,
    W =  -178.278 deg,    P =   -0.030 deg,    R =   -0.998 deg
};
P[393]{
   GP1:
    UF : 0, UT : 6,      CONFIG : 'N U T, 0, 0, 0',
    X =  237.816  mm,    Y =   -3.541  mm,    Z =   674.871  mm,
    W =  -178.460 deg,    P =   -0.027 deg,    R =   -0.998 deg
};
P[394]{
   GP1:
    UF : 0, UT : 6,      CONFIG : 'N U T, 0, 0, 0',
    X =  238.058  mm,    Y =   1.943  mm,    Z =   675.235  mm,
    W =  -178.752 deg,    P =   -0.022 deg,    R =   -0.999 deg
};
P[395]{
   GP1:
    UF : 0, UT : 6,      CONFIG : 'N U T, 0, 0, 0',
    X =  238.024  mm,    Y =   9.530  mm,    Z =   676.209  mm,
    W =  -179.203 deg,    P =   -0.014 deg,    R =   -0.999 deg
};
P[396]{
   GP1:
    UF : 0, UT : 6,      CONFIG : 'N U T, 0, 0, 0',
    X =  238.443  mm,    Y =   14.120  mm,    Z =   676.600  mm,
    W =  -179.411 deg,    P =   -0.010 deg,    R =   -1.000 deg
};
P[397]{
   GP1:
    UF : 0, UT : 6,      CONFIG : 'N U T, 0, 0, 0',
    X =  237.743  mm,    Y =   17.526  mm,    Z =   677.166  mm,
    W =  -179.739 deg,    P =   -0.005 deg,    R =   -1.000 deg
};
P[398]{
   GP1:
    UF : 0, UT : 6,      CONFIG : 'N U T, 0, 0, 0',
    X =  237.873  mm,    Y =   22.373  mm,    Z =   677.478  mm,
    W =  -180.048 deg,    P =   0.001 deg,    R =   -1.000 deg
};
P[399]{
   GP1:
    UF : 0, UT : 6,      CONFIG : 'N U T, 0, 0, 0',
    X =  237.760  mm,    Y =   28.427  mm,    Z =   677.614  mm,
    W =  -180.330 deg,    P =   0.006 deg,    R =   -1.000 deg
};
P[400]{
   GP1:
    UF : 0, UT : 6,      CONFIG : 'N U T, 0, 0, 0',
    X =  237.611  mm,    Y =   34.247  mm,    Z =   677.468  mm,
    W =  -180.661 deg,    P =   0.012 deg,    R =   -1.000 deg
};
P[401]{
   GP1:
    UF : 0, UT : 6,      CONFIG : 'N U T, 0, 0, 0',
    X =  237.278  mm,    Y =   40.465  mm,    Z =   676.904  mm,
    W =  -180.869 deg,    P =   0.015 deg,    R =   -1.000 deg
};
P[402]{
   GP1:
    UF : 0, UT : 6,      CONFIG : 'N U T, 0, 0, 0',
    X =  237.109  mm,    Y =   42.978  mm,    Z =   677.674  mm,
    W =  -180.926 deg,    P =   0.016 deg,    R =   -1.000 deg
};
P[403]{
   GP1:
    UF : 0, UT : 6,      CONFIG : 'N U T, 0, 0, 0',
    X =  237.924  mm,    Y =   46.818  mm,    Z =   676.884  mm,
    W =  -181.027 deg,    P =   0.018 deg,    R =   -1.000 deg
};
P[404]{
   GP1:
    UF : 0, UT : 6,      CONFIG : 'N U T, 0, 0, 0',
    X =  238.005  mm,    Y =   53.855  mm,    Z =   677.512  mm,
    W =  -181.227 deg,    P =   0.021 deg,    R =   -1.000 deg
};
P[405]{
   GP1:
    UF : 0, UT : 6,      CONFIG : 'N U T, 0, 0, 0',
    X =  238.089  mm,    Y =   57.898  mm,    Z =   677.679  mm,
    W =  -181.305 deg,    P =   0.023 deg,    R =   -1.000 deg
};
P[406]{
   GP1:
    UF : 0, UT : 6,      CONFIG : 'N U T, 0, 0, 0',
    X =  237.552  mm,    Y =   62.188  mm,    Z =   677.412  mm,
    W =  -181.342 deg,    P =   0.023 deg,    R =   -1.000 deg
};
P[407]{
   GP1:
    UF : 0, UT : 6,      CONFIG : 'N U T, 0, 0, 0',
    X =  238.039  mm,    Y =   68.846  mm,    Z =   677.586  mm,
    W =  -181.334 deg,    P =   0.023 deg,    R =   -1.000 deg
};
P[408]{
   GP1:
    UF : 0, UT : 6,      CONFIG : 'N U T, 0, 0, 0',
    X =  237.462  mm,    Y =   74.330  mm,    Z =   677.356  mm,
    W =  -181.308 deg,    P =   0.023 deg,    R =   -1.000 deg
};
P[409]{
   GP1:
    UF : 0, UT : 6,      CONFIG : 'N U T, 0, 0, 0',
    X =  238.922  mm,    Y =   78.907  mm,    Z =   677.595  mm,
    W =  -181.269 deg,    P =   0.022 deg,    R =   -1.000 deg
};
P[410]{
   GP1:
    UF : 0, UT : 6,      CONFIG : 'N U T, 0, 0, 0',
    X =  238.350  mm,    Y =   86.026  mm,    Z =   677.232  mm,
    W =  -181.166 deg,    P =   0.020 deg,    R =   -1.000 deg
};
P[411]{
   GP1:
    UF : 0, UT : 6,      CONFIG : 'N U T, 0, 0, 0',
    X =  237.660  mm,    Y =   91.890  mm,    Z =   676.751  mm,
    W =  -181.095 deg,    P =   0.019 deg,    R =   -1.000 deg
};
P[412]{
   GP1:
